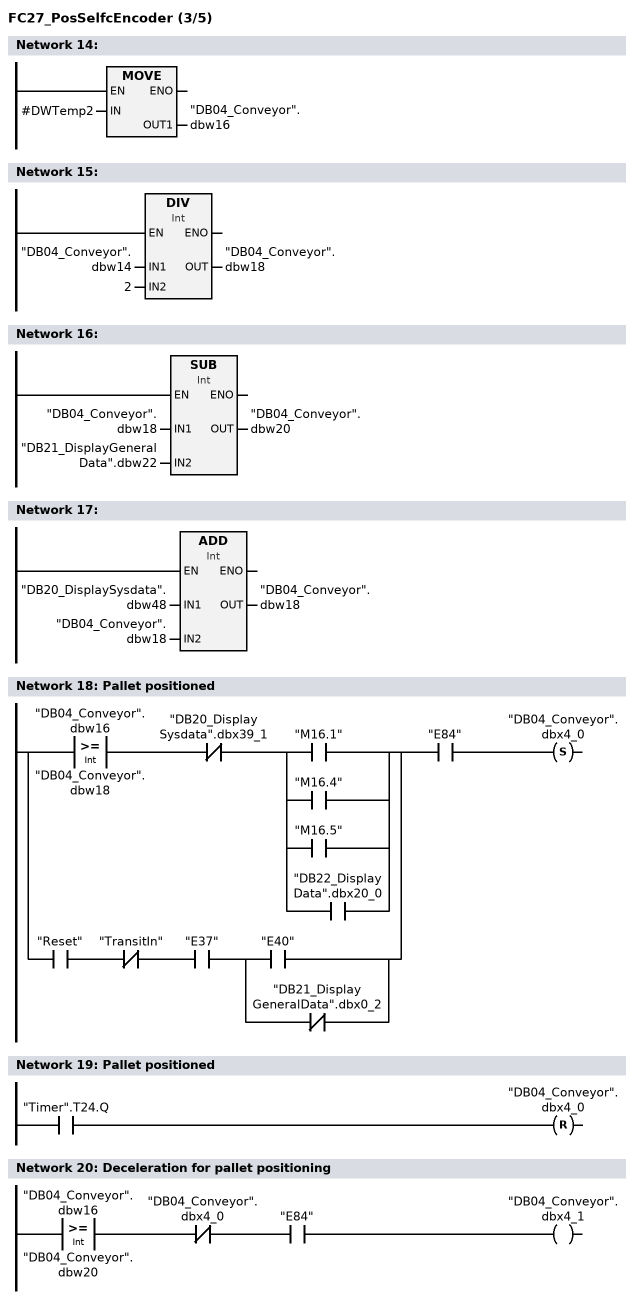
   RUNG wire#powerrail
      { S7_GenerateENO := "TRUE" } Move(in := #DWTemp2, out1 => "DB04_Conveyor".dbw16)
   END_RUNG
   // the same network as SCL:
   "DB04_Conveyor".dbw16 := #DWTemp2;
END_REGION

REGION Network 15
   RUNG wire#powerrail
      { S7_Templates := "SrcType := Int"; S7_GenerateENO := "TRUE" } Div(in1 := "DB04_Conveyor".dbw14, in2 := 2, out => "DB04_Conveyor".dbw18)
   END_RUNG
   // the same network as SCL:
   "DB04_Conveyor".dbw18 := "DB04_Conveyor".dbw14 / 2;
END_REGION

REGION Network 16
   RUNG wire#powerrail
      { S7_Templates := "SrcType := Int"; S7_GenerateENO := "TRUE" } Sub(in1 := "DB04_Conveyor".dbw18, in2 := "DB21_DisplayGeneralData".dbw22, out => "DB04_Conveyor".dbw20)
   END_RUNG
   // the same network as SCL:
   "DB04_Conveyor".dbw20 := "DB04_Conveyor".dbw18 - "DB21_DisplayGeneralData".dbw22;
END_REGION

REGION Network 17
   RUNG wire#powerrail
      { S7_Templates := "SrcType := Int"; S7_GenerateENO := "TRUE" } Add(in1 := "DB20_DisplaySysdata".dbw48, in2 := "DB04_Conveyor".dbw18, out => "DB04_Conveyor".dbw18)
   END_RUNG
   // the same network as SCL:
   "DB04_Conveyor".dbw18 := "DB20_DisplaySysdata".dbw48 + "DB04_Conveyor".dbw18;
END_REGION

REGION Network 18: Pallet positioned
   RUNG wire#powerrail
      { S7_Templates := "SrcType := Int" } GE_Contact(in1 := "DB04_Conveyor".dbw16, in2 := "DB04_Conveyor".dbw18)
      I_Contact( "DB20_DisplaySysdata".dbx39_1 )
      wire#w1
      Contact( "M16.1" )
      wire#w2
      Contact( "E84" )
      S_Coil( "DB04_Conveyor".dbx4_0 )
   END_RUNG
   RUNG wire#w1
      Contact( "M16.4" )
   END_RUNG wire#w2
   RUNG wire#w1
      Contact( "M16.5" )
   END_RUNG wire#w2
   RUNG wire#w1
      Contact( "DB22_DisplayData".dbx20_0 )
   END_RUNG wire#w2
   RUNG wire#powerrail
      Contact( "Reset" )
      I_Contact( "TransitIn" )
      Contact( "E37" )
      wire#w3
      Contact( "E40" )
   END_RUNG wire#w2
   RUNG wire#w3
      I_Contact( "DB21_DisplayGeneralData".dbx0_2 )
   END_RUNG wire#w2
   // the same network as SCL:
   IF ((("DB04_Conveyor".dbw16 >= "DB04_Conveyor".dbw18) AND NOT "DB20_DisplaySysdata".dbx39_1 AND ("M16.1" OR "M16.4" OR "M16.5" OR "DB22_DisplayData".dbx20_0)) OR ("Reset" AND NOT "TransitIn" AND "E37" AND ("E40" OR NOT "DB21_DisplayGeneralData".dbx0_2))) AND "E84" THEN
       "DB04_Conveyor".dbx4_0 := TRUE;
   END_IF;
END_REGION

REGION Network 19: Pallet positioned
   RUNG wire#powerrail
      Contact( "Timer".T24.Q )
      R_Coil( "DB04_Conveyor".dbx4_0 )
   END_RUNG
   // the same network as SCL:
   IF "Timer".T24.Q THEN "DB04_Conveyor".dbx4_0 := FALSE; END_IF;
END_REGION

REGION Network 20: Deceleration for pallet positioning
   RUNG wire#powerrail
      { S7_Templates := "SrcType := Int" } GE_Contact(in1 := "DB04_Conveyor".dbw16, in2 := "DB04_Conveyor".dbw20)
      I_Contact( "DB04_Conveyor".dbx4_0 )
      Contact( "E84" )
      Coil( "DB04_Conveyor".dbx4_1 )
   END_RUNG
   // the same network as SCL:
   "DB04_Conveyor".dbx4_1 := ("DB04_Conveyor".dbw16 >= "DB04_Conveyor".dbw20) AND NOT "DB04_Conveyor".dbx4_0 AND "E84";
END_REGION

REGION Network 21: Short pallet positioned
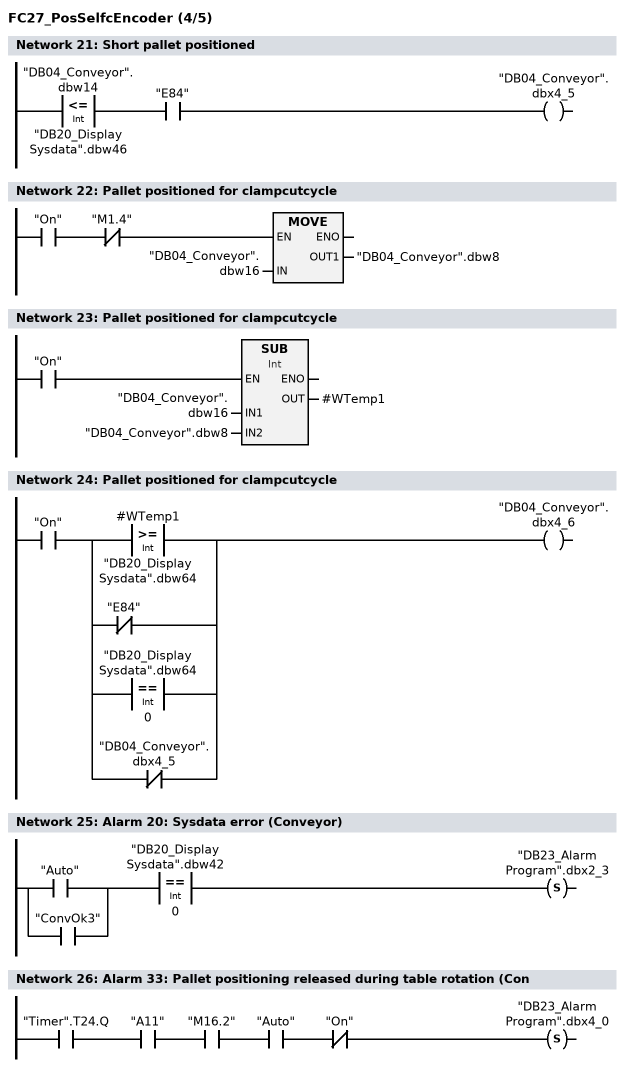
   RUNG wire#powerrail
      { S7_Templates := "SrcType := Int" } LE_Contact(in1 := "DB04_Conveyor".dbw14, in2 := "DB20_DisplaySysdata".dbw46)
      Contact( "E84" )
      Coil( "DB04_Conveyor".dbx4_5 )
   END_RUNG
   // the same network as SCL:
   "DB04_Conveyor".dbx4_5 := ("DB04_Conveyor".dbw14 <= "DB20_DisplaySysdata".dbw46) AND "E84";
END_REGION

REGION Network 22: Pallet positioned for clampcutcycle
   RUNG wire#powerrail
      Contact( "On" )
      I_Contact( "M1.4" )
      { S7_GenerateENO := "TRUE" } Move(in := "DB04_Conveyor".dbw16, out1 => "DB04_Conveyor".dbw8)
   END_RUNG
   // the same network as SCL:
   IF "On" AND NOT "M1.4" THEN "DB04_Conveyor".dbw8 := "DB04_Conveyor".dbw16; END_IF;
END_REGION

REGION Network 23: Pallet positioned for clampcutcycle
   RUNG wire#powerrail
      Contact( "On" )
      { S7_Templates := "SrcType := Int"; S7_GenerateENO := "TRUE" } Sub(in1 := "DB04_Conveyor".dbw16, in2 := "DB04_Conveyor".dbw8, out => #WTemp1)
   END_RUNG
   // the same network as SCL:
   IF "On" THEN #WTemp1 := "DB04_Conveyor".dbw16 - "DB04_Conveyor".dbw8; END_IF;
END_REGION

REGION Network 24: Pallet positioned for clampcutcycle
   RUNG wire#powerrail
      Contact( "On" )
      wire#w1
      { S7_Templates := "SrcType := Int" } GE_Contact(in1 := #WTemp1, in2 := "DB20_DisplaySysdata".dbw64)
      wire#w2
      Coil( "DB04_Conveyor".dbx4_6 )
   END_RUNG
   RUNG wire#w1
      I_Contact( "E84" )
   END_RUNG wire#w2
   RUNG wire#w1
      { S7_Templates := "SrcType := Int" } EQ_Contact(in1 := "DB20_DisplaySysdata".dbw64, in2 := 0)
   END_RUNG wire#w2
   RUNG wire#w1
      I_Contact( "DB04_Conveyor".dbx4_5 )
   END_RUNG wire#w2
   // the same network as SCL:
   "DB04_Conveyor".dbx4_6 := "On" AND ((#WTemp1 >= "DB20_DisplaySysdata".dbw64) OR NOT "E84" OR ("DB20_DisplaySysdata".dbw64 = 0) OR NOT "DB04_Conveyor".dbx4_5);
END_REGION

REGION Network 25: Alarm 20: Sysdata error (Conveyor)
   RUNG wire#powerrail
      Contact( "Auto" )
      wire#w1
      { S7_Templates := "SrcType := Int" } EQ_Contact(in1 := "DB20_DisplaySysdata".dbw42, in2 := 0)
      S_Coil( "DB23_AlarmProgram".dbx2_3 )
   END_RUNG
   RUNG wire#powerrail
      Contact( "ConvOk3" )
   END_RUNG wire#w1
   // the same network as SCL:
   IF ("Auto" OR "ConvOk3") AND ("DB20_DisplaySysdata".dbw42 = 0) THEN
       "DB23_AlarmProgram".dbx2_3 := TRUE;
   END_IF;
END_REGION

REGION Network 26: Alarm 33: Pallet positioning released during table rotation (Con
   RUNG wire#powerrail
      Contact( "Timer".T24.Q )
      Contact( "A11" )
      Contact( "M16.2" )
      Contact( "Auto" )
      I_Contact( "On" )
      S_Coil( "DB23_AlarmProgram".dbx4_0 )
   END_RUNG
   // the same network as SCL:
   IF "Timer".T24.Q AND "A11" AND "M16.2" AND "Auto" AND NOT "On" THEN
       "DB23_AlarmProgram".dbx4_0 := TRUE;
   END_IF;
END_REGION

REGION Network 27: Alarm 36: Wrong pallet positioning (Conveyor)
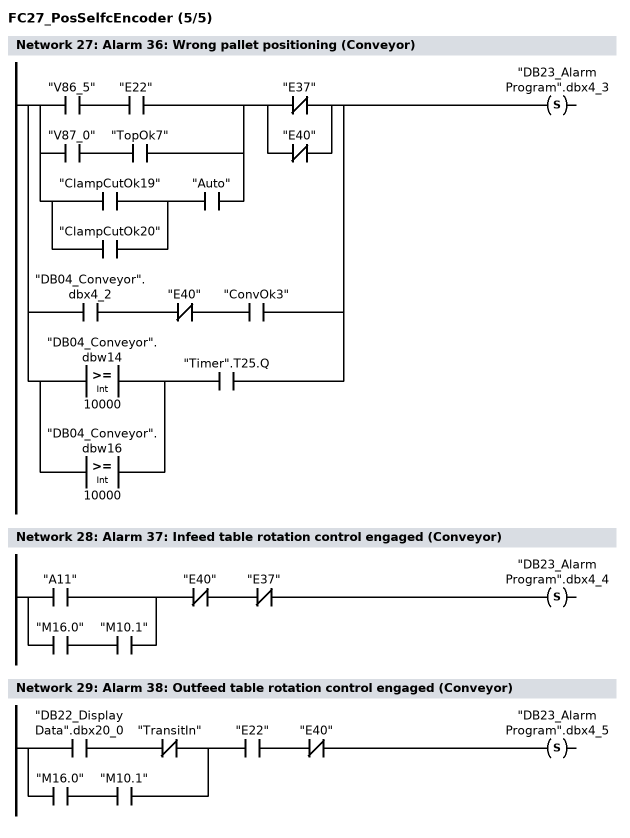
   RUNG wire#powerrail
      Contact( "V86_5" )
      Contact( "E22" )
      wire#w1
      I_Contact( "E37" )
      wire#w3
      S_Coil( "DB23_AlarmProgram".dbx4_3 )
   END_RUNG
   RUNG wire#powerrail
      Contact( "V87_0" )
      Contact( "TopOk7" )
   END_RUNG wire#w1
   RUNG wire#powerrail
      Contact( "ClampCutOk19" )
      wire#w2
      Contact( "Auto" )
   END_RUNG wire#w1
   RUNG wire#powerrail
      Contact( "ClampCutOk20" )
   END_RUNG wire#w2
   RUNG wire#w1
      I_Contact( "E40" )
   END_RUNG wire#w3
   RUNG wire#powerrail
      Contact( "DB04_Conveyor".dbx4_2 )
      I_Contact( "E40" )
      Contact( "ConvOk3" )
   END_RUNG wire#w3
   RUNG wire#powerrail
      { S7_Templates := "SrcType := Int" } GE_Contact(in1 := "DB04_Conveyor".dbw14, in2 := 10000)
      wire#w4
      Contact( "Timer".T25.Q )
   END_RUNG wire#w3
   RUNG wire#powerrail
      { S7_Templates := "SrcType := Int" } GE_Contact(in1 := "DB04_Conveyor".dbw16, in2 := 10000)
   END_RUNG wire#w4
   // the same network as SCL:
   IF ((("V86_5" AND "E22") OR ("V87_0" AND "TopOk7") OR (("ClampCutOk19" OR "ClampCutOk20") AND "Auto")) AND (NOT "E37" OR NOT "E40")) OR ("DB04_Conveyor".dbx4_2 AND NOT "E40" AND "ConvOk3") OR ((("DB04_Conveyor".dbw14 >= 10000) OR ("DB04_Conveyor".dbw16 >= 10000)) AND "Timer".T25.Q) THEN
       "DB23_AlarmProgram".dbx4_3 := TRUE;
   END_IF;
END_REGION

REGION Network 28: Alarm 37: Infeed table rotation control engaged (Conveyor)
   RUNG wire#powerrail
      Contact( "A11" )
      wire#w1
      I_Contact( "E40" )
      I_Contact( "E37" )
      S_Coil( "DB23_AlarmProgram".dbx4_4 )
   END_RUNG
   RUNG wire#powerrail
      Contact( "M16.0" )
      Contact( "M10.1" )
   END_RUNG wire#w1
   // the same network as SCL:
   IF ("A11" OR ("M16.0" AND "M10.1")) AND NOT "E40" AND NOT "E37" THEN
       "DB23_AlarmProgram".dbx4_4 := TRUE;
   END_IF;
END_REGION

REGION Network 29: Alarm 38: Outfeed table rotation control engaged (Conveyor)
   RUNG wire#powerrail
      Contact( "DB22_DisplayData".dbx20_0 )
      I_Contact( "TransitIn" )
      wire#w1
      Contact( "E22" )
      I_Contact( "E40" )
      S_Coil( "DB23_AlarmProgram".dbx4_5 )
   END_RUNG
   RUNG wire#powerrail
      Contact( "M16.0" )
      Contact( "M10.1" )
   END_RUNG wire#w1
   // the same network as SCL:
   IF (("DB22_DisplayData".dbx20_0 AND NOT "TransitIn") OR ("M16.0" AND "M10.1")) AND "E22" AND NOT "E40" THEN
       "DB23_AlarmProgram".dbx4_5 := TRUE;
   END_IF;
END_REGION
END_FUNCTION

FUNCTION "FC31_ConveyorInverter" : Void   // FC31, LAD
TITLE = Conveyor management with inverter
{ S7_Optimized_Access := 'FALSE' }
AUTHOR : Robopac
VERSION : 0.0
// stored: AutoNumber false, IsIECCheckEnabled false, SetENOAutomatically false, UDAEnableTagReadback false
   VAR_TEMP
      TimeUpwardTableCycle : Word;
      TimeUpwardTableCycleInt : Int;
      TempWord : Word;
   END_VAR
   VAR_TEMP   // added for the SCL form of the ladder/FBD networks
      _w1 : Bool;
   END_VAR
BEGIN

REGION Network 1: Timer SA type for conveyor motor
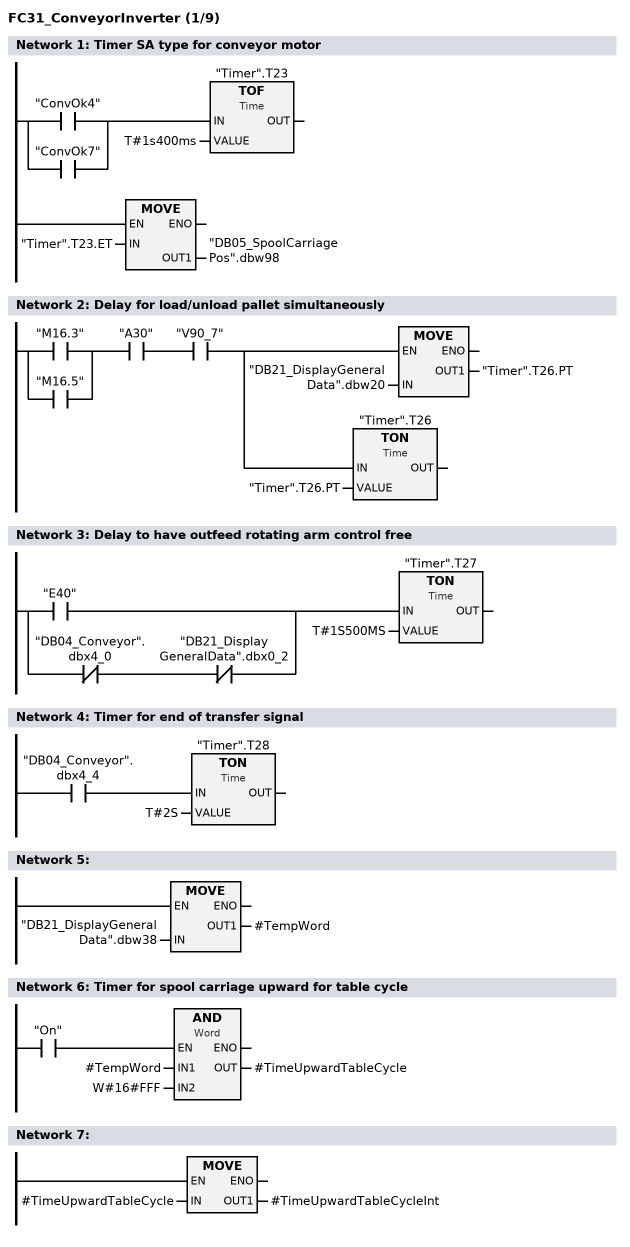
   "Timer".T23.TOF(IN := "ConvOk4" OR "ConvOk7", PT := T#1s400ms);   // TOF coil
   "DB05_SpoolCarriagePos".dbw98 := "Timer".T23.ET;
END_REGION

REGION Network 2: Delay for load/unload pallet simultaneously
   #_w1 := ("M16.3" OR "M16.5") AND "A30" AND "V90_7";
   IF #_w1 THEN "Timer".T26.PT := "DB21_DisplayGeneralData".dbw20; END_IF;
   "Timer".T26.TON(IN := #_w1, PT := "Timer".T26.PT);   // TON coil
END_REGION

REGION Network 3: Delay to have outfeed rotating arm control free
   "Timer".T27.TON(IN := "E40" OR (NOT "DB04_Conveyor".dbx4_0 AND NOT "DB21_DisplayGeneralData".dbx0_2), PT := T#1S500MS);   // TON coil
END_REGION

REGION Network 4: Timer for end of transfer signal
   "Timer".T28.TON(IN := "DB04_Conveyor".dbx4_4, PT := T#2S);   // TON coil
END_REGION

REGION Network 5
   RUNG wire#powerrail
      { S7_GenerateENO := "TRUE" } Move(in := "DB21_DisplayGeneralData".dbw38, out1 => #TempWord)
   END_RUNG
   // the same network as SCL:
   #TempWord := "DB21_DisplayGeneralData".dbw38;
END_REGION

REGION Network 6: Timer for spool carriage upward for table cycle
   RUNG wire#powerrail
      Contact( "On" )
      { S7_Templates := "SrcType := Word"; S7_GenerateENO := "TRUE" } And(in1 := #TempWord, in2 := W#16#FFF, out => #TimeUpwardTableCycle)
   END_RUNG
   // the same network as SCL:
   IF "On" THEN #TimeUpwardTableCycle := #TempWord AND W#16#FFF; END_IF;
END_REGION

REGION Network 7
   RUNG wire#powerrail
      { S7_GenerateENO := "TRUE" } Move(in := #TimeUpwardTableCycle, out1 => #TimeUpwardTableCycleInt)
   END_RUNG
   // the same network as SCL:
   #TimeUpwardTableCycleInt := #TimeUpwardTableCycle;
END_REGION

REGION Network 8: Timer for spool carriage upward for table cycle
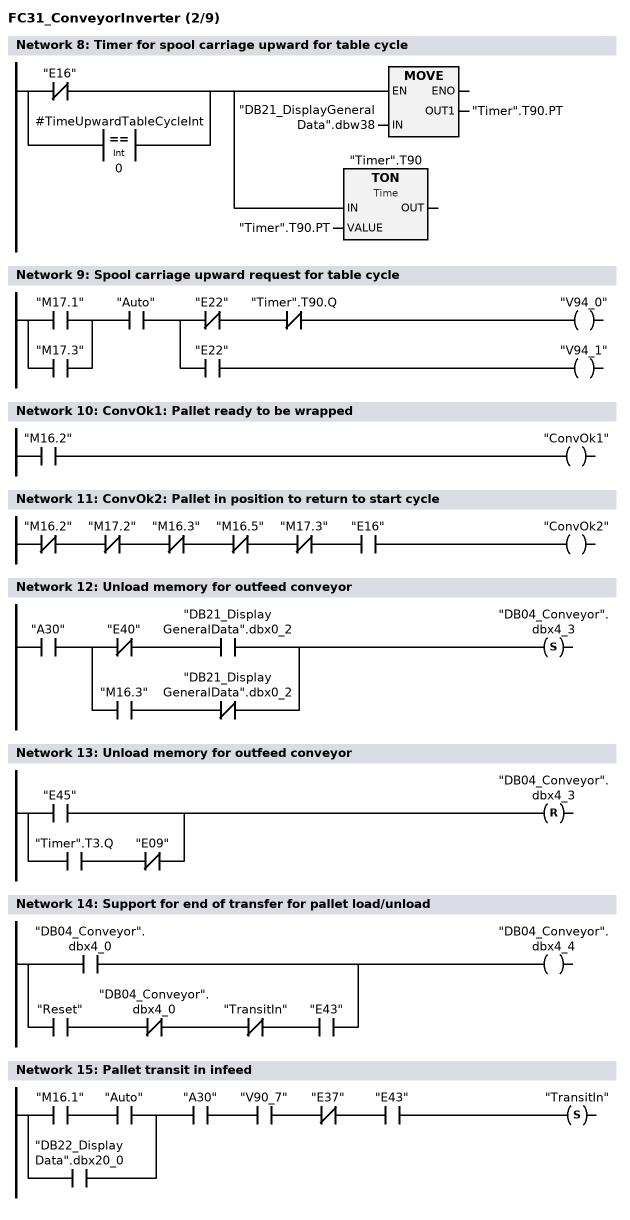
   #_w1 := NOT "E16" OR (#TimeUpwardTableCycleInt = 0);
   IF #_w1 THEN "Timer".T90.PT := "DB21_DisplayGeneralData".dbw38; END_IF;
   "Timer".T90.TON(IN := #_w1, PT := "Timer".T90.PT);   // TON coil
END_REGION

REGION Network 9: Spool carriage upward request for table cycle
   RUNG wire#powerrail
      Contact( "M17.1" )
      wire#w1
      Contact( "Auto" )
      wire#w2
      I_Contact( "E22" )
      I_Contact( "Timer".T90.Q )
      Coil( "V94_0" )
   END_RUNG
   RUNG wire#powerrail
      Contact( "M17.3" )
   END_RUNG wire#w1
   RUNG wire#w2
      Contact( "E22" )
      Coil( "V94_1" )
   END_RUNG
   // the same network as SCL:
   #_w1 := ("M17.1" OR "M17.3") AND "Auto";
   "V94_0" := #_w1 AND NOT "E22" AND NOT "Timer".T90.Q;
   "V94_1" := #_w1 AND "E22";
END_REGION

REGION Network 10: ConvOk1: Pallet ready to be wrapped
   RUNG wire#powerrail
      Contact( "M16.2" )
      Coil( "ConvOk1" )
   END_RUNG
   // the same network as SCL:
   "ConvOk1" := "M16.2";
END_REGION

REGION Network 11: ConvOk2: Pallet in position to return to start cycle
   RUNG wire#powerrail
      I_Contact( "M16.2" )
      I_Contact( "M17.2" )
      I_Contact( "M16.3" )
      I_Contact( "M16.5" )
      I_Contact( "M17.3" )
      Contact( "E16" )
      Coil( "ConvOk2" )
   END_RUNG
   // the same network as SCL:
   "ConvOk2" := NOT "M16.2" AND NOT "M17.2" AND NOT "M16.3" AND NOT "M16.5" AND NOT "M17.3" AND "E16";
END_REGION

REGION Network 12: Unload memory for outfeed conveyor
   RUNG wire#powerrail
      Contact( "A30" )
      wire#w1
      I_Contact( "E40" )
      Contact( "DB21_DisplayGeneralData".dbx0_2 )
      wire#w2
      S_Coil( "DB04_Conveyor".dbx4_3 )
   END_RUNG
   RUNG wire#w1
      Contact( "M16.3" )
      I_Contact( "DB21_DisplayGeneralData".dbx0_2 )
   END_RUNG wire#w2
   // the same network as SCL:
   IF "A30" AND ((NOT "E40" AND "DB21_DisplayGeneralData".dbx0_2) OR ("M16.3" AND NOT "DB21_DisplayGeneralData".dbx0_2)) THEN
       "DB04_Conveyor".dbx4_3 := TRUE;
   END_IF;
END_REGION

REGION Network 13: Unload memory for outfeed conveyor
   RUNG wire#powerrail
      Contact( "E45" )
      wire#w1
      R_Coil( "DB04_Conveyor".dbx4_3 )
   END_RUNG
   RUNG wire#powerrail
      Contact( "Timer".T3.Q )
      I_Contact( "E09" )
   END_RUNG wire#w1
   // the same network as SCL:
   IF "E45" OR ("Timer".T3.Q AND NOT "E09") THEN "DB04_Conveyor".dbx4_3 := FALSE; END_IF;
END_REGION

REGION Network 14: Support for end of transfer for pallet load/unload
   RUNG wire#powerrail
      Contact( "DB04_Conveyor".dbx4_0 )
      wire#w1
      Coil( "DB04_Conveyor".dbx4_4 )
   END_RUNG
   RUNG wire#powerrail
      Contact( "Reset" )
      I_Contact( "DB04_Conveyor".dbx4_0 )
      I_Contact( "TransitIn" )
      Contact( "E43" )
   END_RUNG wire#w1
   // the same network as SCL:
   "DB04_Conveyor".dbx4_4 := "DB04_Conveyor".dbx4_0 OR ("Reset" AND NOT "DB04_Conveyor".dbx4_0 AND NOT "TransitIn" AND "E43");
END_REGION

REGION Network 15: Pallet transit in infeed
   RUNG wire#powerrail
      Contact( "M16.1" )
      Contact( "Auto" )
      wire#w1
      Contact( "A30" )
      Contact( "V90_7" )
      I_Contact( "E37" )
      Contact( "E43" )
      S_Coil( "TransitIn" )
   END_RUNG
   RUNG wire#powerrail
      Contact( "DB22_DisplayData".dbx20_0 )
   END_RUNG wire#w1
   // the same network as SCL:
   IF (("M16.1" AND "Auto") OR "DB22_DisplayData".dbx20_0) AND "A30" AND "V90_7" AND NOT "E37" AND "E43" THEN
       "TransitIn" := TRUE;
   END_IF;
END_REGION

REGION Network 16: Pallet transit in infeed
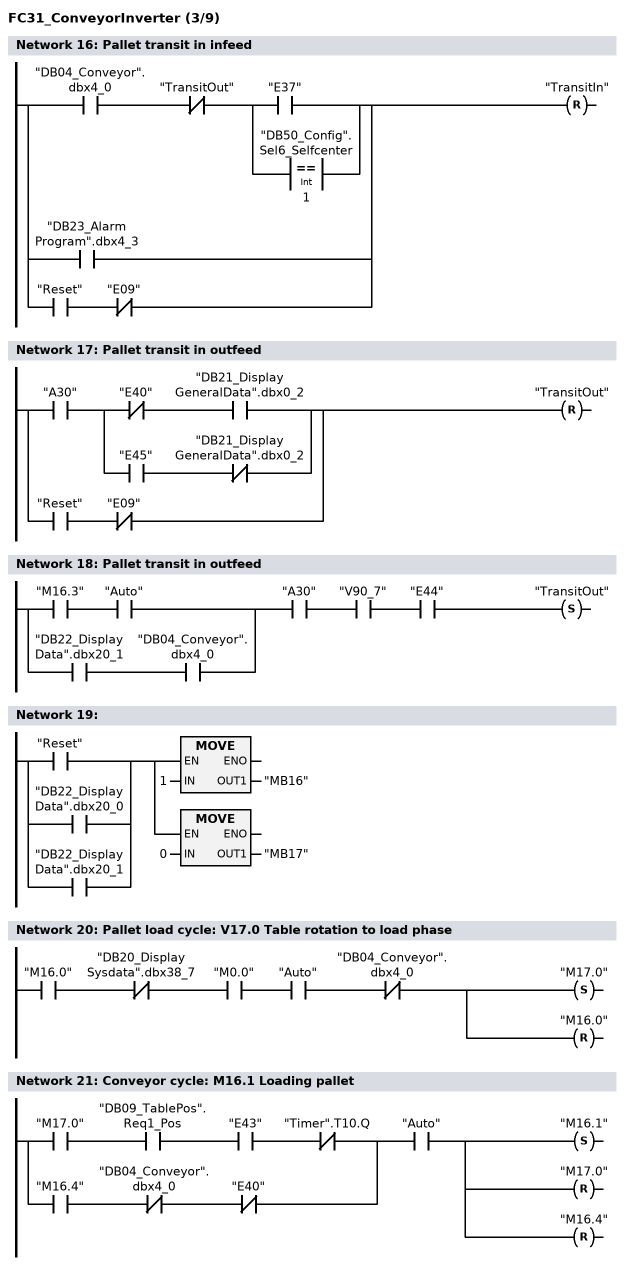
   IF ("DB04_Conveyor".dbx4_0 AND NOT "TransitOut" AND (("DB50_Config".Sel6_Selfcenter = 1) OR "E37")) OR "DB23_AlarmProgram".dbx4_3 OR ("Reset" AND NOT "E09") THEN
       "TransitIn" := FALSE;
   END_IF;
END_REGION

REGION Network 17: Pallet transit in outfeed
   RUNG wire#powerrail
      Contact( "A30" )
      wire#w1
      I_Contact( "E40" )
      Contact( "DB21_DisplayGeneralData".dbx0_2 )
      wire#w2
      R_Coil( "TransitOut" )
   END_RUNG
   RUNG wire#w1
      Contact( "E45" )
      I_Contact( "DB21_DisplayGeneralData".dbx0_2 )
   END_RUNG wire#w2
   RUNG wire#powerrail
      Contact( "Reset" )
      I_Contact( "E09" )
   END_RUNG wire#w2
   // the same network as SCL:
   IF ("A30" AND ((NOT "E40" AND "DB21_DisplayGeneralData".dbx0_2) OR ("E45" AND NOT "DB21_DisplayGeneralData".dbx0_2))) OR ("Reset" AND NOT "E09") THEN
       "TransitOut" := FALSE;
   END_IF;
END_REGION

REGION Network 18: Pallet transit in outfeed
   RUNG wire#powerrail
      Contact( "M16.3" )
      Contact( "Auto" )
      wire#w1
      Contact( "A30" )
      Contact( "V90_7" )
      Contact( "E44" )
      S_Coil( "TransitOut" )
   END_RUNG
   RUNG wire#powerrail
      Contact( "DB22_DisplayData".dbx20_1 )
      Contact( "DB04_Conveyor".dbx4_0 )
   END_RUNG wire#w1
   // the same network as SCL:
   IF (("M16.3" AND "Auto") OR ("DB22_DisplayData".dbx20_1 AND "DB04_Conveyor".dbx4_0)) AND "A30" AND "V90_7" AND "E44" THEN
       "TransitOut" := TRUE;
   END_IF;
END_REGION

REGION Network 19
   RUNG wire#powerrail
      Contact( "Reset" )
      wire#w1
      { S7_GenerateENO := "TRUE" } Move(in := 1, out1 => "MB16")
   END_RUNG
   RUNG wire#powerrail
      Contact( "DB22_DisplayData".dbx20_0 )
   END_RUNG wire#w1
   RUNG wire#powerrail
      Contact( "DB22_DisplayData".dbx20_1 )
   END_RUNG wire#w1
   RUNG wire#w1
      { S7_GenerateENO := "TRUE" } Move(in := 0, out1 => "MB17")
   END_RUNG
   // the same network as SCL:
   IF "Reset" OR "DB22_DisplayData".dbx20_0 OR "DB22_DisplayData".dbx20_1 THEN
       "MB16" := 1;
       "MB17" := 0;
   END_IF;
END_REGION

REGION Network 20: Pallet load cycle: V17.0 Table rotation to load phase
   RUNG wire#powerrail
      Contact( "M16.0" )
      I_Contact( "DB20_DisplaySysdata".dbx38_7 )
      Contact( "M0.0" )
      Contact( "Auto" )
      I_Contact( "DB04_Conveyor".dbx4_0 )
      wire#w1
      S_Coil( "M17.0" )
   END_RUNG
   RUNG wire#w1
      R_Coil( "M16.0" )
   END_RUNG
   // the same network as SCL:
   IF "M16.0" AND NOT "DB20_DisplaySysdata".dbx38_7 AND "M0.0" AND "Auto" AND NOT "DB04_Conveyor".dbx4_0 THEN
       "M17.0" := TRUE;
       "M16.0" := FALSE;
   END_IF;
END_REGION

REGION Network 21: Conveyor cycle: M16.1 Loading pallet
   RUNG wire#powerrail
      Contact( "M17.0" )
      Contact( "DB09_TablePos".Req1_Pos )
      Contact( "E43" )
      I_Contact( "Timer".T10.Q )
      wire#w1
      Contact( "Auto" )
      wire#w2
      S_Coil( "M16.1" )
   END_RUNG
   RUNG wire#powerrail
      Contact( "M16.4" )
      I_Contact( "DB04_Conveyor".dbx4_0 )
      I_Contact( "E40" )
   END_RUNG wire#w1
   RUNG wire#w2
      R_Coil( "M17.0" )
   END_RUNG
   RUNG wire#w2
      R_Coil( "M16.4" )
   END_RUNG
   // the same network as SCL:
   IF (("M17.0" AND "DB09_TablePos".Req1_Pos AND "E43" AND NOT "Timer".T10.Q) OR ("M16.4" AND NOT "DB04_Conveyor".dbx4_0 AND NOT "E40")) AND "Auto" THEN
       "M16.1" := TRUE;
   END_IF;
   #_w1 := (("M17.0" AND "DB09_TablePos".Req1_Pos AND "E43" AND NOT "Timer".T10.Q) OR ("M16.4" AND NOT "DB04_Conveyor".dbx4_0 AND NOT "E40")) AND "Auto";
   IF #_w1 THEN
       "M17.0" := FALSE;
       "M16.4" := FALSE;
   END_IF;
END_REGION

REGION Network 22: Pallet load cycle: V17.1 Table rotation to machine phase from lo
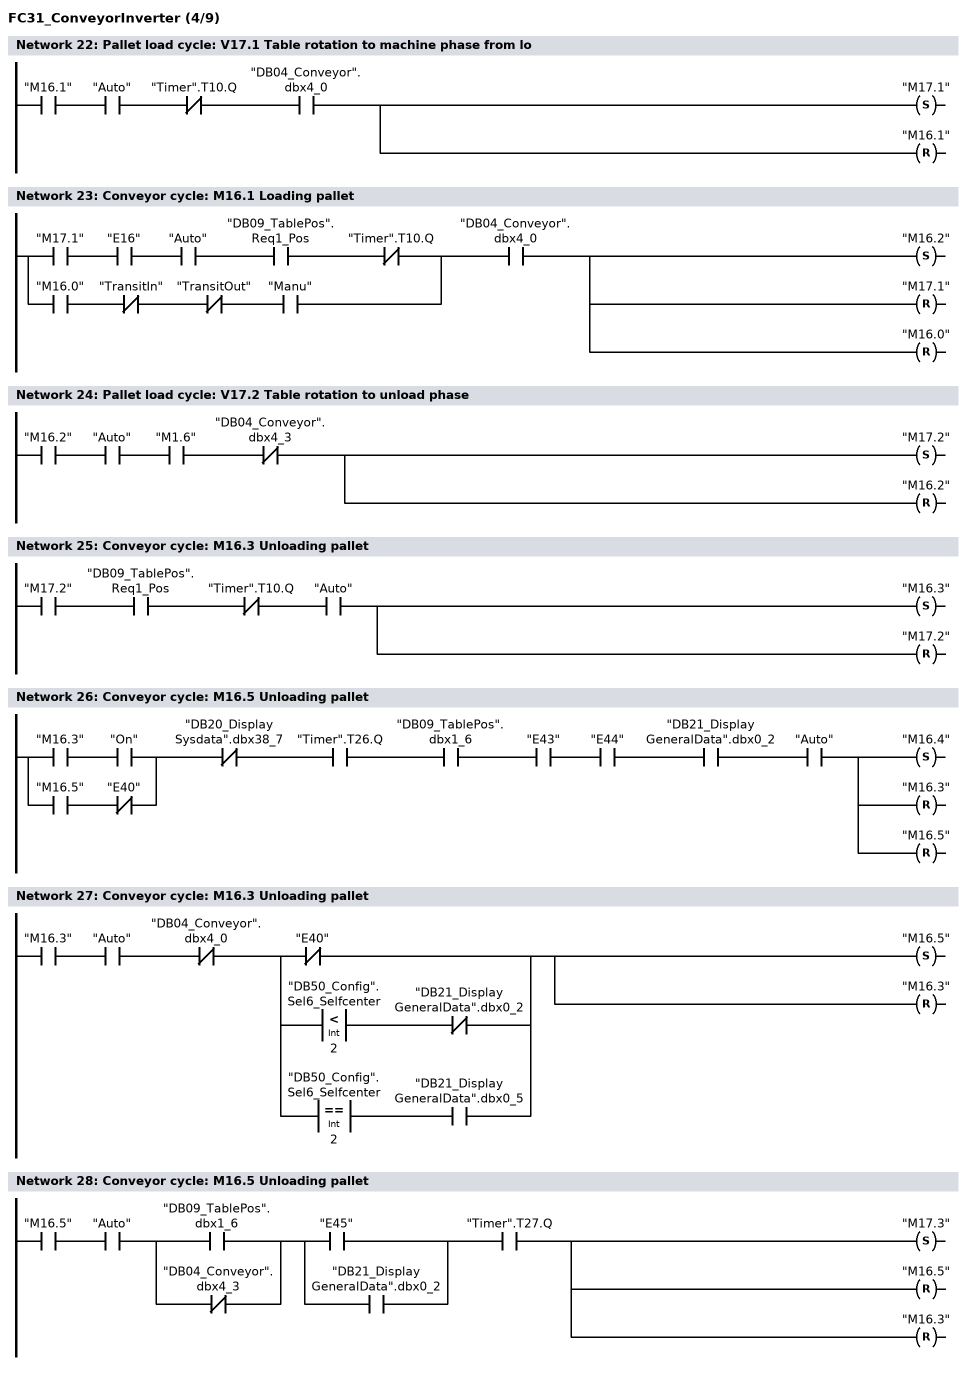
   RUNG wire#powerrail
      Contact( "M16.1" )
      Contact( "Auto" )
      I_Contact( "Timer".T10.Q )
      Contact( "DB04_Conveyor".dbx4_0 )
      wire#w1
      S_Coil( "M17.1" )
   END_RUNG
   RUNG wire#w1
      R_Coil( "M16.1" )
   END_RUNG
   // the same network as SCL:
   IF "M16.1" AND "Auto" AND NOT "Timer".T10.Q AND "DB04_Conveyor".dbx4_0 THEN
       "M17.1" := TRUE;
       "M16.1" := FALSE;
   END_IF;
END_REGION

REGION Network 23: Conveyor cycle: M16.1 Loading pallet
   RUNG wire#powerrail
      Contact( "M17.1" )
      Contact( "E16" )
      Contact( "Auto" )
      Contact( "DB09_TablePos".Req1_Pos )
      I_Contact( "Timer".T10.Q )
      wire#w1
      Contact( "DB04_Conveyor".dbx4_0 )
      wire#w2
      S_Coil( "M16.2" )
   END_RUNG
   RUNG wire#powerrail
      Contact( "M16.0" )
      I_Contact( "TransitIn" )
      I_Contact( "TransitOut" )
      Contact( "Manu" )
   END_RUNG wire#w1
   RUNG wire#w2
      R_Coil( "M17.1" )
   END_RUNG
   RUNG wire#w2
      R_Coil( "M16.0" )
   END_RUNG
   // the same network as SCL:
   IF (("M17.1" AND "E16" AND "Auto" AND "DB09_TablePos".Req1_Pos AND NOT "Timer".T10.Q) OR ("M16.0" AND NOT "TransitIn" AND NOT "TransitOut" AND "Manu")) AND "DB04_Conveyor".dbx4_0 THEN
       "M16.2" := TRUE;
   END_IF;
   #_w1 := (("M17.1" AND "E16" AND "Auto" AND "DB09_TablePos".Req1_Pos AND NOT "Timer".T10.Q) OR ("M16.0" AND NOT "TransitIn" AND NOT "TransitOut" AND "Manu")) AND "DB04_Conveyor".dbx4_0;
   IF #_w1 THEN
       "M17.1" := FALSE;
       "M16.0" := FALSE;
   END_IF;
END_REGION

REGION Network 24: Pallet load cycle: V17.2 Table rotation to unload phase
   RUNG wire#powerrail
      Contact( "M16.2" )
      Contact( "Auto" )
      Contact( "M1.6" )
      I_Contact( "DB04_Conveyor".dbx4_3 )
      wire#w1
      S_Coil( "M17.2" )
   END_RUNG
   RUNG wire#w1
      R_Coil( "M16.2" )
   END_RUNG
   // the same network as SCL:
   IF "M16.2" AND "Auto" AND "M1.6" AND NOT "DB04_Conveyor".dbx4_3 THEN
       "M17.2" := TRUE;
       "M16.2" := FALSE;
   END_IF;
END_REGION

REGION Network 25: Conveyor cycle: M16.3 Unloading pallet
   RUNG wire#powerrail
      Contact( "M17.2" )
      Contact( "DB09_TablePos".Req1_Pos )
      I_Contact( "Timer".T10.Q )
      Contact( "Auto" )
      wire#w1
      S_Coil( "M16.3" )
   END_RUNG
   RUNG wire#w1
      R_Coil( "M17.2" )
   END_RUNG
   // the same network as SCL:
   IF "M17.2" AND "DB09_TablePos".Req1_Pos AND NOT "Timer".T10.Q AND "Auto" THEN
       "M16.3" := TRUE;
       "M17.2" := FALSE;
   END_IF;
END_REGION

REGION Network 26: Conveyor cycle: M16.5 Unloading pallet
   RUNG wire#powerrail
      Contact( "M16.3" )
      Contact( "On" )
      wire#w1
      I_Contact( "DB20_DisplaySysdata".dbx38_7 )
      Contact( "Timer".T26.Q )
      Contact( "DB09_TablePos".dbx1_6 )
      Contact( "E43" )
      Contact( "E44" )
      Contact( "DB21_DisplayGeneralData".dbx0_2 )
      Contact( "Auto" )
      wire#w2
      S_Coil( "M16.4" )
   END_RUNG
   RUNG wire#powerrail
      Contact( "M16.5" )
      I_Contact( "E40" )
   END_RUNG wire#w1
   RUNG wire#w2
      R_Coil( "M16.3" )
   END_RUNG
   RUNG wire#w2
      R_Coil( "M16.5" )
   END_RUNG
   // the same network as SCL:
   IF (("M16.3" AND "On") OR ("M16.5" AND NOT "E40")) AND NOT "DB20_DisplaySysdata".dbx38_7 AND "Timer".T26.Q AND "DB09_TablePos".dbx1_6 AND "E43" AND "E44" AND "DB21_DisplayGeneralData".dbx0_2 AND "Auto" THEN
       "M16.4" := TRUE;
   END_IF;
   #_w1 := (("M16.3" AND "On") OR ("M16.5" AND NOT "E40")) AND NOT "DB20_DisplaySysdata".dbx38_7 AND "Timer".T26.Q AND "DB09_TablePos".dbx1_6 AND "E43" AND "E44" AND "DB21_DisplayGeneralData".dbx0_2 AND "Auto";
   IF #_w1 THEN
       "M16.3" := FALSE;
       "M16.5" := FALSE;
   END_IF;
END_REGION

REGION Network 27: Conveyor cycle: M16.3 Unloading pallet
   RUNG wire#powerrail
      Contact( "M16.3" )
      Contact( "Auto" )
      I_Contact( "DB04_Conveyor".dbx4_0 )
      wire#w1
      I_Contact( "E40" )
      wire#w2
      S_Coil( "M16.5" )
   END_RUNG
   RUNG wire#w1
      { S7_Templates := "SrcType := Int" } LT_Contact(in1 := "DB50_Config".Sel6_Selfcenter, in2 := 2)
      I_Contact( "DB21_DisplayGeneralData".dbx0_2 )
   END_RUNG wire#w2
   RUNG wire#w1
      { S7_Templates := "SrcType := Int" } EQ_Contact(in1 := "DB50_Config".Sel6_Selfcenter, in2 := 2)
      Contact( "DB21_DisplayGeneralData".dbx0_5 )
   END_RUNG wire#w2
   RUNG wire#w2
      R_Coil( "M16.3" )
   END_RUNG
   // the same network as SCL:
   IF "M16.3" AND "Auto" AND NOT "DB04_Conveyor".dbx4_0 AND (NOT "E40" OR (("DB50_Config".Sel6_Selfcenter < 2) AND NOT "DB21_DisplayGeneralData".dbx0_2) OR (("DB50_Config".Sel6_Selfcenter = 2) AND "DB21_DisplayGeneralData".dbx0_5)) THEN
       "M16.5" := TRUE;
       "M16.3" := FALSE;
   END_IF;
END_REGION

REGION Network 28: Conveyor cycle: M16.5 Unloading pallet
   RUNG wire#powerrail
      Contact( "M16.5" )
      Contact( "Auto" )
      wire#w1
      Contact( "DB09_TablePos".dbx1_6 )
      wire#w2
      Contact( "E45" )
      wire#w3
      Contact( "Timer".T27.Q )
      wire#w4
      S_Coil( "M17.3" )
   END_RUNG
   RUNG wire#w1
      I_Contact( "DB04_Conveyor".dbx4_3 )
   END_RUNG wire#w2
   RUNG wire#w2
      Contact( "DB21_DisplayGeneralData".dbx0_2 )
   END_RUNG wire#w3
   RUNG wire#w4
      R_Coil( "M16.5" )
   END_RUNG
   RUNG wire#w4
      R_Coil( "M16.3" )
   END_RUNG
   // the same network as SCL:
   IF "M16.5" AND "Auto" AND ("DB09_TablePos".dbx1_6 OR NOT "DB04_Conveyor".dbx4_3) AND ("E45" OR "DB21_DisplayGeneralData".dbx0_2) AND "Timer".T27.Q THEN
       "M17.3" := TRUE;
   END_IF;
   #_w1 := "M16.5" AND "Auto" AND ("DB09_TablePos".dbx1_6 OR NOT "DB04_Conveyor".dbx4_3) AND ("E45" OR "DB21_DisplayGeneralData".dbx0_2) AND "Timer".T27.Q;
   IF #_w1 THEN
       "M16.5" := FALSE;
       "M16.3" := FALSE;
   END_IF;
END_REGION

REGION Network 29: Conveyor cycle: M16.0 Start cycle
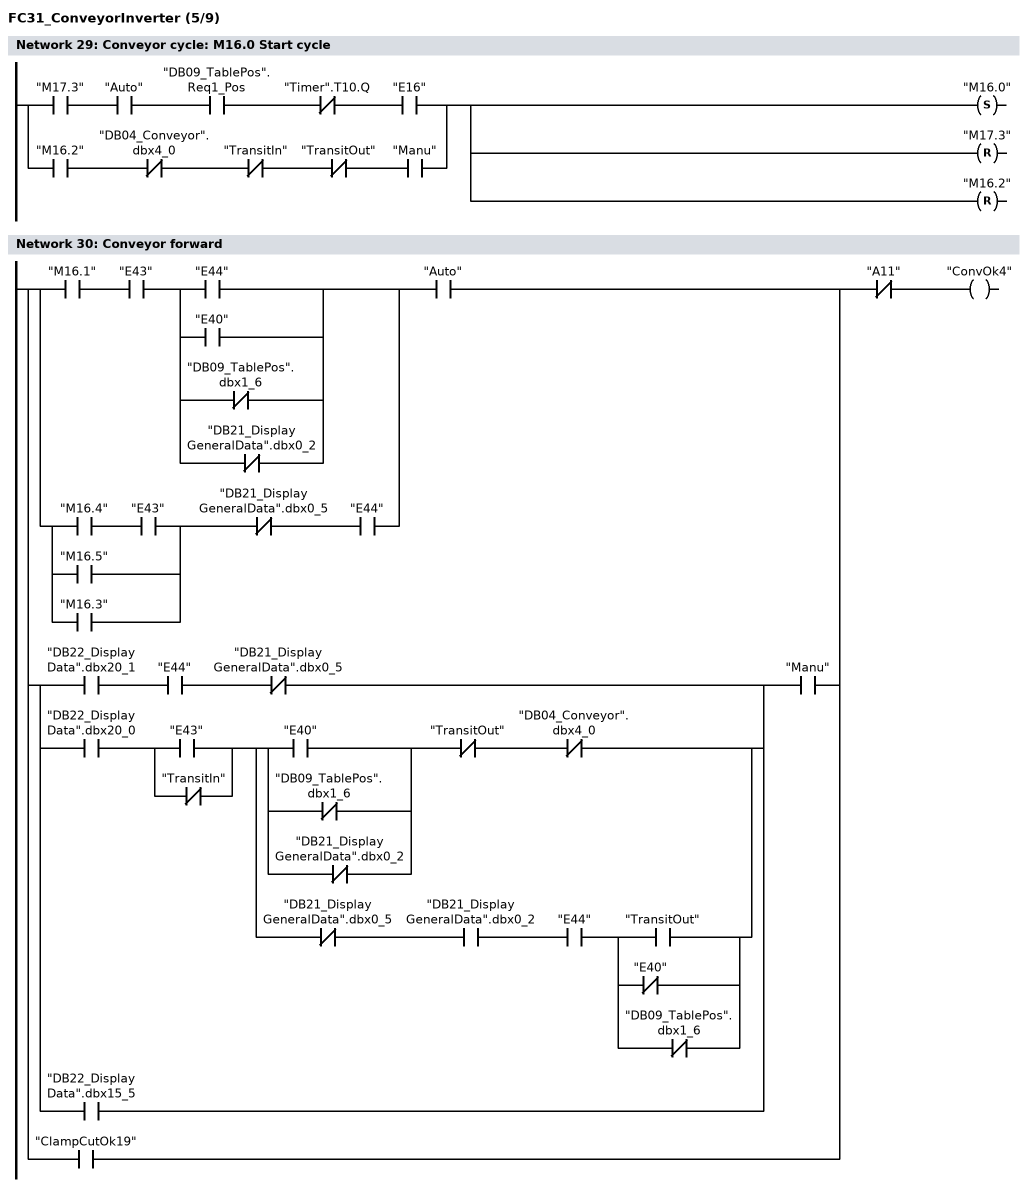
   RUNG wire#powerrail
      Contact( "M17.3" )
      Contact( "Auto" )
      Contact( "DB09_TablePos".Req1_Pos )
      I_Contact( "Timer".T10.Q )
      Contact( "E16" )
      wire#w1
      S_Coil( "M16.0" )
   END_RUNG
   RUNG wire#powerrail
      Contact( "M16.2" )
      I_Contact( "DB04_Conveyor".dbx4_0 )
      I_Contact( "TransitIn" )
      I_Contact( "TransitOut" )
      Contact( "Manu" )
   END_RUNG wire#w1
   RUNG wire#w1
      R_Coil( "M17.3" )
   END_RUNG
   RUNG wire#w1
      R_Coil( "M16.2" )
   END_RUNG
   // the same network as SCL:
   IF ("M17.3" AND "Auto" AND "DB09_TablePos".Req1_Pos AND NOT "Timer".T10.Q AND "E16") OR ("M16.2" AND NOT "DB04_Conveyor".dbx4_0 AND NOT "TransitIn" AND NOT "TransitOut" AND "Manu") THEN
       "M16.0" := TRUE;
   END_IF;
   #_w1 := ("M17.3" AND "Auto" AND "DB09_TablePos".Req1_Pos AND NOT "Timer".T10.Q AND "E16") OR ("M16.2" AND NOT "DB04_Conveyor".dbx4_0 AND NOT "TransitIn" AND NOT "TransitOut" AND "Manu");
   IF #_w1 THEN
       "M17.3" := FALSE;
       "M16.2" := FALSE;
   END_IF;
END_REGION

REGION Network 30: Conveyor forward
   RUNG wire#powerrail
      Contact( "M16.1" )
      Contact( "E43" )
      wire#w1
      Contact( "E44" )
      wire#w2
      Contact( "Auto" )
      wire#w4
      I_Contact( "A11" )
      Coil( "ConvOk4" )
   END_RUNG
   RUNG wire#w1
      Contact( "E40" )
   END_RUNG wire#w2
   RUNG wire#w1
      I_Contact( "DB09_TablePos".dbx1_6 )
   END_RUNG wire#w2
   RUNG wire#w1
      I_Contact( "DB21_DisplayGeneralData".dbx0_2 )
   END_RUNG wire#w2
   RUNG wire#powerrail
      Contact( "M16.4" )
      Contact( "E43" )
      wire#w3
      I_Contact( "DB21_DisplayGeneralData".dbx0_5 )
      Contact( "E44" )
   END_RUNG wire#w2
   RUNG wire#powerrail
      Contact( "M16.5" )
   END_RUNG wire#w3
   RUNG wire#powerrail
      Contact( "M16.3" )
   END_RUNG wire#w3
   RUNG wire#powerrail
      Contact( "DB22_DisplayData".dbx20_1 )
      Contact( "E44" )
      I_Contact( "DB21_DisplayGeneralData".dbx0_5 )
      wire#w5
      Contact( "Manu" )
   END_RUNG wire#w4
   RUNG wire#powerrail
      Contact( "DB22_DisplayData".dbx20_0 )
      wire#w6
      Contact( "E43" )
      wire#w7
      Contact( "E40" )
      wire#w8
      I_Contact( "TransitOut" )
      I_Contact( "DB04_Conveyor".dbx4_0 )
   END_RUNG wire#w5
   RUNG wire#w6
      I_Contact( "TransitIn" )
   END_RUNG wire#w7
   RUNG wire#w7
      I_Contact( "DB09_TablePos".dbx1_6 )
   END_RUNG wire#w8
   RUNG wire#w7
      I_Contact( "DB21_DisplayGeneralData".dbx0_2 )
   END_RUNG wire#w8
   RUNG wire#w7
      I_Contact( "DB21_DisplayGeneralData".dbx0_5 )
      Contact( "DB21_DisplayGeneralData".dbx0_2 )
      Contact( "E44" )
      wire#w9
      Contact( "TransitOut" )
   END_RUNG wire#w5
   RUNG wire#w9
      I_Contact( "E40" )
   END_RUNG wire#w5
   RUNG wire#w9
      I_Contact( "DB09_TablePos".dbx1_6 )
   END_RUNG wire#w5
   RUNG wire#powerrail
      Contact( "DB22_DisplayData".dbx15_5 )
   END_RUNG wire#w5
   RUNG wire#powerrail
      Contact( "ClampCutOk19" )
   END_RUNG wire#w4
   // the same network as SCL:
   "ConvOk4" := (((("M16.1" AND "E43" AND ("E44" OR "E40" OR NOT "DB09_TablePos".dbx1_6 OR NOT "DB21_DisplayGeneralData".dbx0_2)) OR ((("M16.4" AND "E43") OR "M16.5" OR "M16.3") AND NOT "DB21_DisplayGeneralData".dbx0_5 AND "E44")) AND "Auto") OR ((("DB22_DisplayData".dbx20_1 AND "E44" AND NOT "DB21_DisplayGeneralData".dbx0_5) OR ("DB22_DisplayData".dbx20_0 AND ("E43" OR NOT "TransitIn") AND ((("E40" OR NOT "DB09_TablePos".dbx1_6 OR NOT "DB21_DisplayGeneralData".dbx0_2) AND NOT "TransitOut" AND NOT "DB04_Conveyor".dbx4_0) OR (NOT "DB21_DisplayGeneralData".dbx0_5 AND "DB21_DisplayGeneralData".dbx0_2 AND "E44" AND ("TransitOut" OR NOT "E40" OR NOT "DB09_TablePos".dbx1_6)))) OR "DB22_DisplayData".dbx15_5) AND "Manu") OR "ClampCutOk19") AND NOT "A11";
END_REGION

REGION Network 31: ConvOk7: Backward for inverter
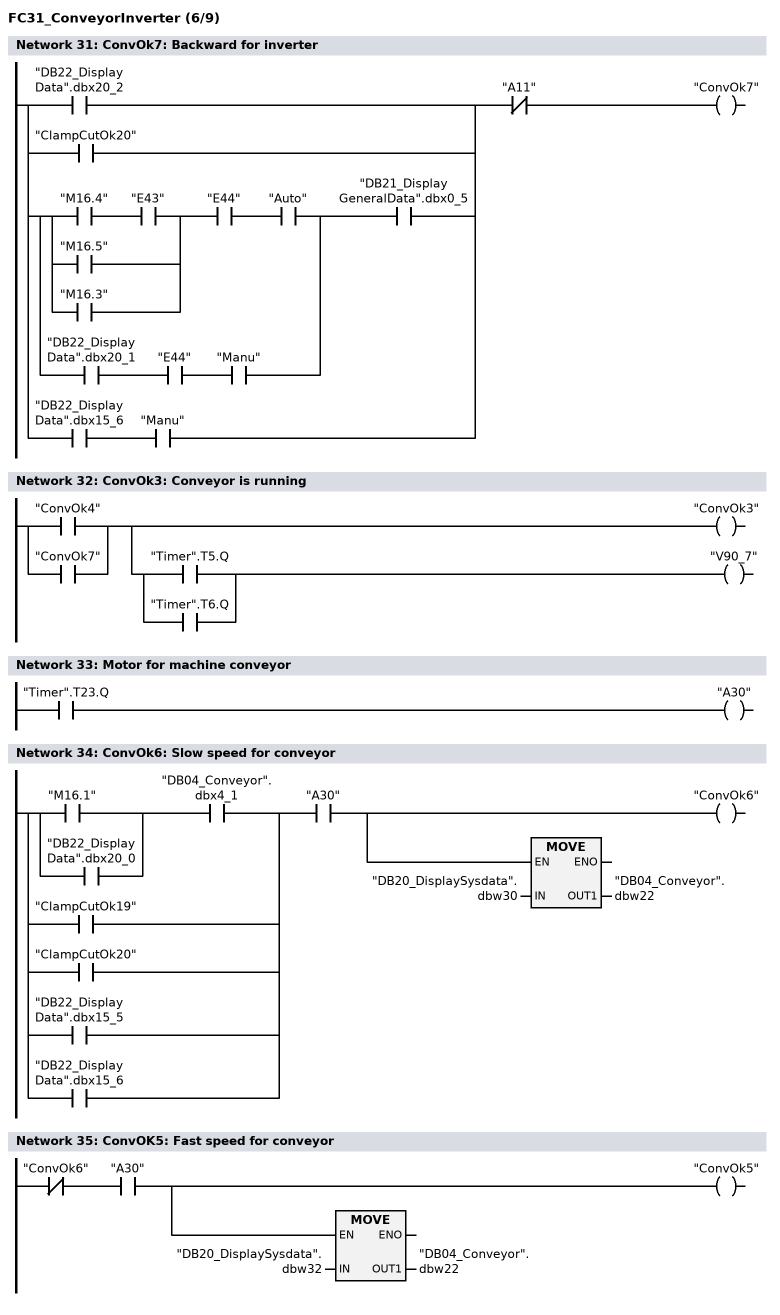
   RUNG wire#powerrail
      Contact( "DB22_DisplayData".dbx20_2 )
      wire#w1
      I_Contact( "A11" )
      Coil( "ConvOk7" )
   END_RUNG
   RUNG wire#powerrail
      Contact( "ClampCutOk20" )
   END_RUNG wire#w1
   RUNG wire#powerrail
      Contact( "M16.4" )
      Contact( "E43" )
      wire#w2
      Contact( "E44" )
      Contact( "Auto" )
      wire#w3
      Contact( "DB21_DisplayGeneralData".dbx0_5 )
   END_RUNG wire#w1
   RUNG wire#powerrail
      Contact( "M16.5" )
   END_RUNG wire#w2
   RUNG wire#powerrail
      Contact( "M16.3" )
   END_RUNG wire#w2
   RUNG wire#powerrail
      Contact( "DB22_DisplayData".dbx20_1 )
      Contact( "E44" )
      Contact( "Manu" )
   END_RUNG wire#w3
   RUNG wire#powerrail
      Contact( "DB22_DisplayData".dbx15_6 )
      Contact( "Manu" )
   END_RUNG wire#w1
   // the same network as SCL:
   "ConvOk7" := ("DB22_DisplayData".dbx20_2 OR "ClampCutOk20" OR ((((("M16.4" AND "E43") OR "M16.5" OR "M16.3") AND "E44" AND "Auto") OR ("DB22_DisplayData".dbx20_1 AND "E44" AND "Manu")) AND "DB21_DisplayGeneralData".dbx0_5) OR ("DB22_DisplayData".dbx15_6 AND "Manu")) AND NOT "A11";
END_REGION

REGION Network 32: ConvOk3: Conveyor is running
   RUNG wire#powerrail
      Contact( "ConvOk4" )
      wire#w1
      Coil( "ConvOk3" )
   END_RUNG
   RUNG wire#powerrail
      Contact( "ConvOk7" )
   END_RUNG wire#w1
   RUNG wire#w1
      Contact( "Timer".T5.Q )
      wire#w2
      Coil( "V90_7" )
   END_RUNG
   RUNG wire#w1
      Contact( "Timer".T6.Q )
   END_RUNG wire#w2
   // the same network as SCL:
   "ConvOk3" := "ConvOk4" OR "ConvOk7";
   "V90_7" := "ConvOk3" AND ("Timer".T5.Q OR "Timer".T6.Q);
END_REGION

REGION Network 33: Motor for machine conveyor
   RUNG wire#powerrail
      Contact( "Timer".T23.Q )
      Coil( "A30" )
   END_RUNG
   // the same network as SCL:
   "A30" := "Timer".T23.Q;
END_REGION

REGION Network 34: ConvOk6: Slow speed for conveyor
   RUNG wire#powerrail
      Contact( "M16.1" )
      wire#w1
      Contact( "DB04_Conveyor".dbx4_1 )
      wire#w2
      Contact( "A30" )
      wire#w3
      Coil( "ConvOk6" )
   END_RUNG
   RUNG wire#powerrail
      Contact( "DB22_DisplayData".dbx20_0 )
   END_RUNG wire#w1
   RUNG wire#powerrail
      Contact( "ClampCutOk19" )
   END_RUNG wire#w2
   RUNG wire#powerrail
      Contact( "ClampCutOk20" )
   END_RUNG wire#w2
   RUNG wire#powerrail
      Contact( "DB22_DisplayData".dbx15_5 )
   END_RUNG wire#w2
   RUNG wire#powerrail
      Contact( "DB22_DisplayData".dbx15_6 )
   END_RUNG wire#w2
   RUNG wire#w3
      { S7_GenerateENO := "TRUE" } Move(in := "DB20_DisplaySysdata".dbw30, out1 => "DB04_Conveyor".dbw22)
   END_RUNG
   // the same network as SCL:
   "ConvOk6" := ((("M16.1" OR "DB22_DisplayData".dbx20_0) AND "DB04_Conveyor".dbx4_1) OR "ClampCutOk19" OR "ClampCutOk20" OR "DB22_DisplayData".dbx15_5 OR "DB22_DisplayData".dbx15_6) AND "A30";
   IF "ConvOk6" THEN "DB04_Conveyor".dbw22 := "DB20_DisplaySysdata".dbw30; END_IF;
END_REGION

REGION Network 35: ConvOK5: Fast speed for conveyor
   RUNG wire#powerrail
      I_Contact( "ConvOk6" )
      Contact( "A30" )
      wire#w1
      Coil( "ConvOk5" )
   END_RUNG
   RUNG wire#w1
      { S7_GenerateENO := "TRUE" } Move(in := "DB20_DisplaySysdata".dbw32, out1 => "DB04_Conveyor".dbw22)
   END_RUNG
   // the same network as SCL:
   "ConvOk5" := NOT "ConvOk6" AND "A30";
   IF "ConvOk5" THEN "DB04_Conveyor".dbw22 := "DB20_DisplaySysdata".dbw32; END_IF;
END_REGION

REGION Network 36: rotation inverter: Support for speed selection
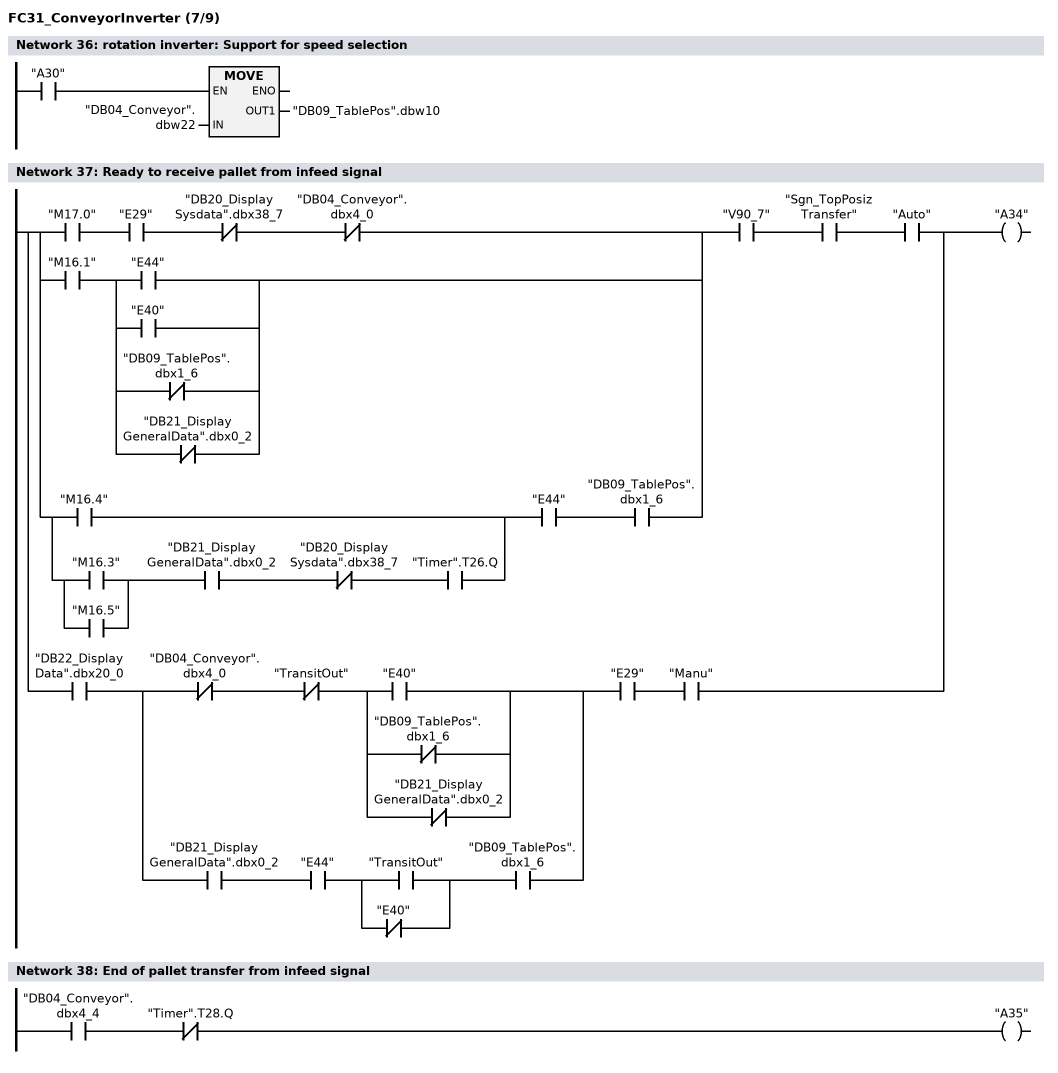
   RUNG wire#powerrail
      Contact( "A30" )
      { S7_GenerateENO := "TRUE" } Move(in := "DB04_Conveyor".dbw22, out1 => "DB09_TablePos".dbw10)
   END_RUNG
   // the same network as SCL:
   IF "A30" THEN "DB09_TablePos".dbw10 := "DB04_Conveyor".dbw22; END_IF;
END_REGION

REGION Network 37: Ready to receive pallet from infeed signal
   RUNG wire#powerrail
      Contact( "M17.0" )
      Contact( "E29" )
      I_Contact( "DB20_DisplaySysdata".dbx38_7 )
      I_Contact( "DB04_Conveyor".dbx4_0 )
      wire#w1
      Contact( "V90_7" )
      Contact( "Sgn_TopPosizTransfer" )
      Contact( "Auto" )
      wire#w5
      Coil( "A34" )
   END_RUNG
   RUNG wire#powerrail
      Contact( "M16.1" )
      wire#w2
      Contact( "E44" )
   END_RUNG wire#w1
   RUNG wire#w2
      Contact( "E40" )
   END_RUNG wire#w1
   RUNG wire#w2
      I_Contact( "DB09_TablePos".dbx1_6 )
   END_RUNG wire#w1
   RUNG wire#w2
      I_Contact( "DB21_DisplayGeneralData".dbx0_2 )
   END_RUNG wire#w1
   RUNG wire#powerrail
      Contact( "M16.4" )
      wire#w3
      Contact( "E44" )
      Contact( "DB09_TablePos".dbx1_6 )
   END_RUNG wire#w1
   RUNG wire#powerrail
      Contact( "M16.3" )
      wire#w4
      Contact( "DB21_DisplayGeneralData".dbx0_2 )
      I_Contact( "DB20_DisplaySysdata".dbx38_7 )
      Contact( "Timer".T26.Q )
   END_RUNG wire#w3
   RUNG wire#powerrail
      Contact( "M16.5" )
   END_RUNG wire#w4
   RUNG wire#powerrail
      Contact( "DB22_DisplayData".dbx20_0 )
      wire#w6
      I_Contact( "DB04_Conveyor".dbx4_0 )
      I_Contact( "TransitOut" )
      wire#w7
      Contact( "E40" )
      wire#w8
      Contact( "E29" )
      Contact( "Manu" )
   END_RUNG wire#w5
   RUNG wire#w7
      I_Contact( "DB09_TablePos".dbx1_6 )
   END_RUNG wire#w8
   RUNG wire#w7
      I_Contact( "DB21_DisplayGeneralData".dbx0_2 )
   END_RUNG wire#w8
   RUNG wire#w6
      Contact( "DB21_DisplayGeneralData".dbx0_2 )
      Contact( "E44" )
      wire#w9
      Contact( "TransitOut" )
      wire#w10
      Contact( "DB09_TablePos".dbx1_6 )
   END_RUNG wire#w8
   RUNG wire#w9
      I_Contact( "E40" )
   END_RUNG wire#w10
   // the same network as SCL:
   "A34" := ((("M17.0" AND "E29" AND NOT "DB20_DisplaySysdata".dbx38_7 AND NOT "DB04_Conveyor".dbx4_0) OR ("M16.1" AND ("E44" OR "E40" OR NOT "DB09_TablePos".dbx1_6 OR NOT "DB21_DisplayGeneralData".dbx0_2)) OR (("M16.4" OR (("M16.3" OR "M16.5") AND "DB21_DisplayGeneralData".dbx0_2 AND NOT "DB20_DisplaySysdata".dbx38_7 AND "Timer".T26.Q)) AND "E44" AND "DB09_TablePos".dbx1_6)) AND "V90_7" AND "Sgn_TopPosizTransfer" AND "Auto") OR ("DB22_DisplayData".dbx20_0 AND ((NOT "DB04_Conveyor".dbx4_0 AND NOT "TransitOut" AND ("E40" OR NOT "DB09_TablePos".dbx1_6 OR NOT "DB21_DisplayGeneralData".dbx0_2)) OR ("DB21_DisplayGeneralData".dbx0_2 AND "E44" AND ("TransitOut" OR NOT "E40") AND "DB09_TablePos".dbx1_6)) AND "E29" AND "Manu");
END_REGION

REGION Network 38: End of pallet transfer from infeed signal
   RUNG wire#powerrail
      Contact( "DB04_Conveyor".dbx4_4 )
      I_Contact( "Timer".T28.Q )
      Coil( "A35" )
   END_RUNG
   // the same network as SCL:
   "A35" := "DB04_Conveyor".dbx4_4 AND NOT "Timer".T28.Q;
END_REGION

REGION Network 39: Pallet ready for outfeed signal
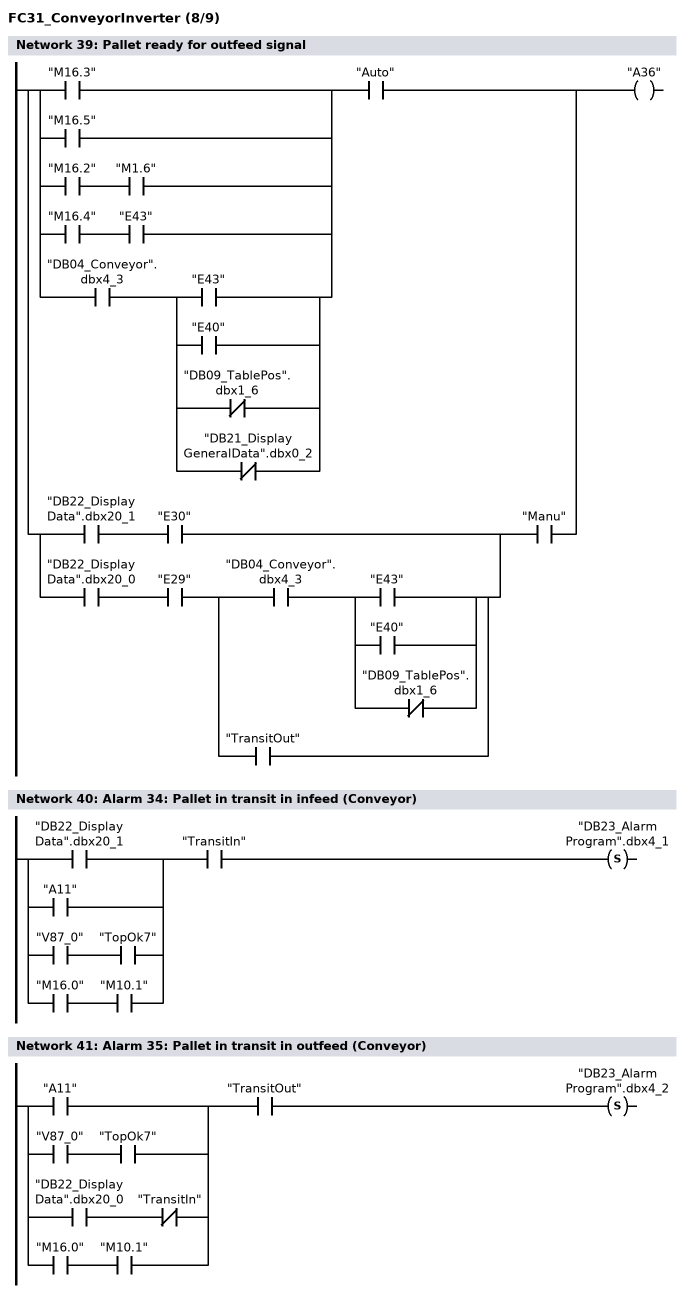
   RUNG wire#powerrail
      Contact( "M16.3" )
      wire#w1
      Contact( "Auto" )
      wire#w3
      Coil( "A36" )
   END_RUNG
   RUNG wire#powerrail
      Contact( "M16.5" )
   END_RUNG wire#w1
   RUNG wire#powerrail
      Contact( "M16.2" )
      Contact( "M1.6" )
   END_RUNG wire#w1
   RUNG wire#powerrail
      Contact( "M16.4" )
      Contact( "E43" )
   END_RUNG wire#w1
   RUNG wire#powerrail
      Contact( "DB04_Conveyor".dbx4_3 )
      wire#w2
      Contact( "E43" )
   END_RUNG wire#w1
   RUNG wire#w2
      Contact( "E40" )
   END_RUNG wire#w1
   RUNG wire#w2
      I_Contact( "DB09_TablePos".dbx1_6 )
   END_RUNG wire#w1
   RUNG wire#w2
      I_Contact( "DB21_DisplayGeneralData".dbx0_2 )
   END_RUNG wire#w1
   RUNG wire#powerrail
      Contact( "DB22_DisplayData".dbx20_1 )
      Contact( "E30" )
      wire#w4
      Contact( "Manu" )
   END_RUNG wire#w3
   RUNG wire#powerrail
      Contact( "DB22_DisplayData".dbx20_0 )
      Contact( "E29" )
      wire#w5
      Contact( "DB04_Conveyor".dbx4_3 )
      wire#w6
      Contact( "E43" )
   END_RUNG wire#w4
   RUNG wire#w6
      Contact( "E40" )
   END_RUNG wire#w4
   RUNG wire#w6
      I_Contact( "DB09_TablePos".dbx1_6 )
   END_RUNG wire#w4
   RUNG wire#w5
      Contact( "TransitOut" )
   END_RUNG wire#w4
   // the same network as SCL:
   "A36" := (("M16.3" OR "M16.5" OR ("M16.2" AND "M1.6") OR ("M16.4" AND "E43") OR ("DB04_Conveyor".dbx4_3 AND ("E43" OR "E40" OR NOT "DB09_TablePos".dbx1_6 OR NOT "DB21_DisplayGeneralData".dbx0_2))) AND "Auto") OR ((("DB22_DisplayData".dbx20_1 AND "E30") OR ("DB22_DisplayData".dbx20_0 AND "E29" AND (("DB04_Conveyor".dbx4_3 AND ("E43" OR "E40" OR NOT "DB09_TablePos".dbx1_6)) OR "TransitOut"))) AND "Manu");
END_REGION

REGION Network 40: Alarm 34: Pallet in transit in infeed (Conveyor)
   RUNG wire#powerrail
      Contact( "DB22_DisplayData".dbx20_1 )
      wire#w1
      Contact( "TransitIn" )
      S_Coil( "DB23_AlarmProgram".dbx4_1 )
   END_RUNG
   RUNG wire#powerrail
      Contact( "A11" )
   END_RUNG wire#w1
   RUNG wire#powerrail
      Contact( "V87_0" )
      Contact( "TopOk7" )
   END_RUNG wire#w1
   RUNG wire#powerrail
      Contact( "M16.0" )
      Contact( "M10.1" )
   END_RUNG wire#w1
   // the same network as SCL:
   IF ("DB22_DisplayData".dbx20_1 OR "A11" OR ("V87_0" AND "TopOk7") OR ("M16.0" AND "M10.1")) AND "TransitIn" THEN
       "DB23_AlarmProgram".dbx4_1 := TRUE;
   END_IF;
END_REGION

REGION Network 41: Alarm 35: Pallet in transit in outfeed (Conveyor)
   RUNG wire#powerrail
      Contact( "A11" )
      wire#w1
      Contact( "TransitOut" )
      S_Coil( "DB23_AlarmProgram".dbx4_2 )
   END_RUNG
   RUNG wire#powerrail
      Contact( "V87_0" )
      Contact( "TopOk7" )
   END_RUNG wire#w1
   RUNG wire#powerrail
      Contact( "DB22_DisplayData".dbx20_0 )
      I_Contact( "TransitIn" )
   END_RUNG wire#w1
   RUNG wire#powerrail
      Contact( "M16.0" )
      Contact( "M10.1" )
   END_RUNG wire#w1
   // the same network as SCL:
   IF ("A11" OR ("V87_0" AND "TopOk7") OR ("DB22_DisplayData".dbx20_0 AND NOT "TransitIn") OR ("M16.0" AND "M10.1")) AND "TransitOut" THEN
       "DB23_AlarmProgram".dbx4_2 := TRUE;
   END_IF;
END_REGION

REGION Network 42: Alarm 39: Technoplat table not in load phase
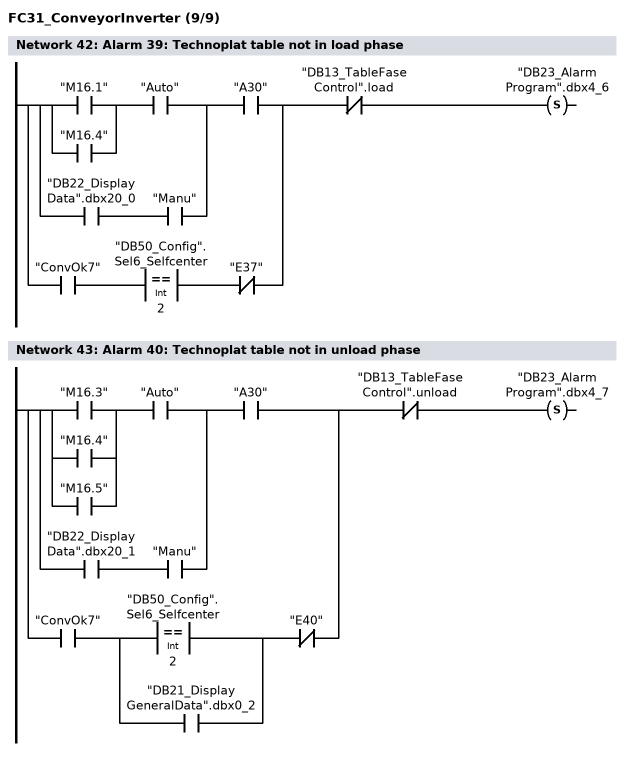
   RUNG wire#powerrail
      Contact( "M16.1" )
      wire#w1
      Contact( "Auto" )
      wire#w2
      Contact( "A30" )
      wire#w3
      I_Contact( "DB13_TableFaseControl".load )
      S_Coil( "DB23_AlarmProgram".dbx4_6 )
   END_RUNG
   RUNG wire#powerrail
      Contact( "M16.4" )
   END_RUNG wire#w1
   RUNG wire#powerrail
      Contact( "DB22_DisplayData".dbx20_0 )
      Contact( "Manu" )
   END_RUNG wire#w2
   RUNG wire#powerrail
      Contact( "ConvOk7" )
      { S7_Templates := "SrcType := Int" } EQ_Contact(in1 := "DB50_Config".Sel6_Selfcenter, in2 := 2)
      I_Contact( "E37" )
   END_RUNG wire#w3
   // the same network as SCL:
   IF ((((("M16.1" OR "M16.4") AND "Auto") OR ("DB22_DisplayData".dbx20_0 AND "Manu")) AND "A30") OR ("ConvOk7" AND ("DB50_Config".Sel6_Selfcenter = 2) AND NOT "E37")) AND NOT "DB13_TableFaseControl".load THEN
       "DB23_AlarmProgram".dbx4_6 := TRUE;
   END_IF;
END_REGION

REGION Network 43: Alarm 40: Technoplat table not in unload phase
   RUNG wire#powerrail
      Contact( "M16.3" )
      wire#w1
      Contact( "Auto" )
      wire#w2
      Contact( "A30" )
      wire#w3
      I_Contact( "DB13_TableFaseControl".unload )
      S_Coil( "DB23_AlarmProgram".dbx4_7 )
   END_RUNG
   RUNG wire#powerrail
      Contact( "M16.4" )
   END_RUNG wire#w1
   RUNG wire#powerrail
      Contact( "M16.5" )
   END_RUNG wire#w1
   RUNG wire#powerrail
      Contact( "DB22_DisplayData".dbx20_1 )
      Contact( "Manu" )
   END_RUNG wire#w2
   RUNG wire#powerrail
      Contact( "ConvOk7" )
      wire#w4
      { S7_Templates := "SrcType := Int" } EQ_Contact(in1 := "DB50_Config".Sel6_Selfcenter, in2 := 2)
      wire#w5
      I_Contact( "E40" )
   END_RUNG wire#w3
   RUNG wire#w4
      Contact( "DB21_DisplayGeneralData".dbx0_2 )
   END_RUNG wire#w5
   // the same network as SCL:
   IF ((((("M16.3" OR "M16.4" OR "M16.5") AND "Auto") OR ("DB22_DisplayData".dbx20_1 AND "Manu")) AND "A30") OR ("ConvOk7" AND (("DB50_Config".Sel6_Selfcenter = 2) OR "DB21_DisplayGeneralData".dbx0_2) AND NOT "E40")) AND NOT "DB13_TableFaseControl".unload THEN
       "DB23_AlarmProgram".dbx4_7 := TRUE;
   END_IF;
END_REGION
END_FUNCTION

FUNCTION "FC86_Conveyor_5_IN_3_OUT" : Void   // FC86, LAD
TITLE = Conveyor_5_IN_3_OUT
{ S7_Optimized_Access := 'TRUE' }
VERSION : 0.1
// 5+3 (Fitembal)
// stored: AutoNumber false, IsIECCheckEnabled false, SetENOAutomatically false, UDAEnableTagReadback false
   VAR_TEMP   // added for the SCL form of the ladder/FBD networks
      _w1 : Bool;
      _w2 : Bool;
   END_VAR
BEGIN

REGION Network 1: Manual operation for conveyor
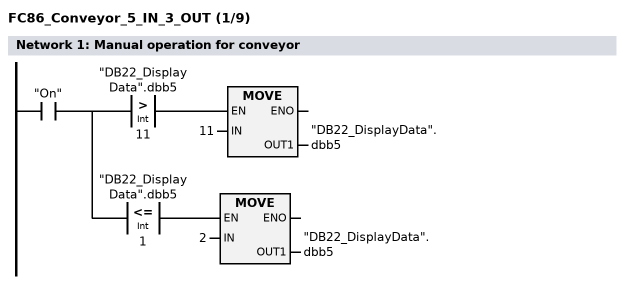
   RUNG wire#powerrail
      Contact( "On" )
      wire#w1
      { S7_Templates := "SrcType := Int" } GT_Contact(in1 := "DB22_DisplayData".dbb5, in2 := 11)
      { S7_GenerateENO := "TRUE" } Move(in := 11, out1 => "DB22_DisplayData".dbb5)
   END_RUNG
   RUNG wire#w1
      { S7_Templates := "SrcType := Int" } LE_Contact(in1 := "DB22_DisplayData".dbb5, in2 := 1)
      { S7_GenerateENO := "TRUE" } Move(in := 2, out1 => "DB22_DisplayData".dbb5)
   END_RUNG
   // the same network as SCL:
   IF "On" AND ("DB22_DisplayData".dbb5 > 11) THEN "DB22_DisplayData".dbb5 := 11; END_IF;
   IF "On" AND ("DB22_DisplayData".dbb5 <= 1) THEN "DB22_DisplayData".dbb5 := 2; END_IF;
END_REGION

REGION Network 2: Manual operation for conveyor
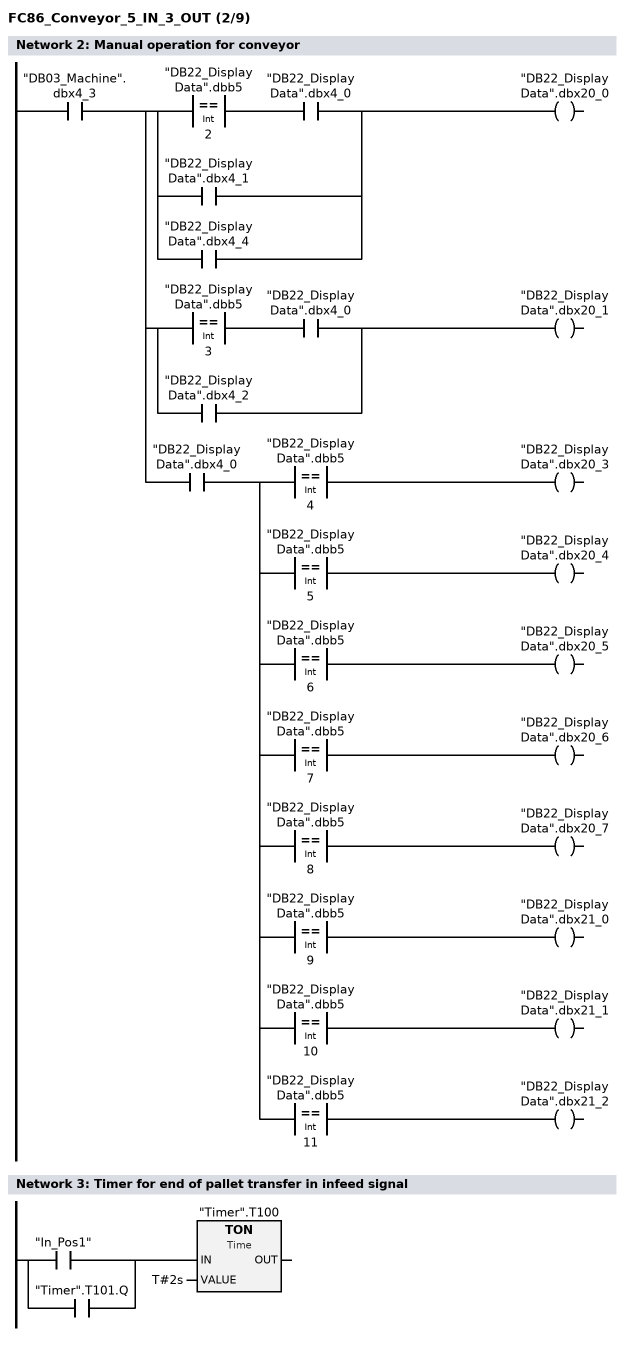
   RUNG wire#powerrail
      Contact( "DB03_Machine".dbx4_3 )
      wire#w1
      { S7_Templates := "SrcType := Int" } EQ_Contact(in1 := "DB22_DisplayData".dbb5, in2 := 2)
      Contact( "DB22_DisplayData".dbx4_0 )
      wire#w2
      Coil( "DB22_DisplayData".dbx20_0 )
   END_RUNG
   RUNG wire#w1
      Contact( "DB22_DisplayData".dbx4_1 )
   END_RUNG wire#w2
   RUNG wire#w1
      Contact( "DB22_DisplayData".dbx4_4 )
   END_RUNG wire#w2
   RUNG wire#w1
      { S7_Templates := "SrcType := Int" } EQ_Contact(in1 := "DB22_DisplayData".dbb5, in2 := 3)
      Contact( "DB22_DisplayData".dbx4_0 )
      wire#w3
      Coil( "DB22_DisplayData".dbx20_1 )
   END_RUNG
   RUNG wire#w1
      Contact( "DB22_DisplayData".dbx4_2 )
   END_RUNG wire#w3
   RUNG wire#w1
      Contact( "DB22_DisplayData".dbx4_0 )
      wire#w4
      { S7_Templates := "SrcType := Int" } EQ_Contact(in1 := "DB22_DisplayData".dbb5, in2 := 4)
      Coil( "DB22_DisplayData".dbx20_3 )
   END_RUNG
   RUNG wire#w4
      { S7_Templates := "SrcType := Int" } EQ_Contact(in1 := "DB22_DisplayData".dbb5, in2 := 5)
      Coil( "DB22_DisplayData".dbx20_4 )
   END_RUNG
   RUNG wire#w4
      { S7_Templates := "SrcType := Int" } EQ_Contact(in1 := "DB22_DisplayData".dbb5, in2 := 6)
      Coil( "DB22_DisplayData".dbx20_5 )
   END_RUNG
   RUNG wire#w4
      { S7_Templates := "SrcType := Int" } EQ_Contact(in1 := "DB22_DisplayData".dbb5, in2 := 7)
      Coil( "DB22_DisplayData".dbx20_6 )
   END_RUNG
   RUNG wire#w4
      { S7_Templates := "SrcType := Int" } EQ_Contact(in1 := "DB22_DisplayData".dbb5, in2 := 8)
      Coil( "DB22_DisplayData".dbx20_7 )
   END_RUNG
   RUNG wire#w4
      { S7_Templates := "SrcType := Int" } EQ_Contact(in1 := "DB22_DisplayData".dbb5, in2 := 9)
      Coil( "DB22_DisplayData".dbx21_0 )
   END_RUNG
   RUNG wire#w4
      { S7_Templates := "SrcType := Int" } EQ_Contact(in1 := "DB22_DisplayData".dbb5, in2 := 10)
      Coil( "DB22_DisplayData".dbx21_1 )
   END_RUNG
   RUNG wire#w4
      { S7_Templates := "SrcType := Int" } EQ_Contact(in1 := "DB22_DisplayData".dbb5, in2 := 11)
      Coil( "DB22_DisplayData".dbx21_2 )
   END_RUNG
   // the same network as SCL:
   "DB22_DisplayData".dbx20_0 := "DB03_Machine".dbx4_3 AND ((("DB22_DisplayData".dbb5 = 2) AND "DB22_DisplayData".dbx4_0) OR "DB22_DisplayData".dbx4_1 OR "DB22_DisplayData".dbx4_4);
   "DB22_DisplayData".dbx20_1 := "DB03_Machine".dbx4_3 AND ((("DB22_DisplayData".dbb5 = 3) AND "DB22_DisplayData".dbx4_0) OR "DB22_DisplayData".dbx4_2);
   #_w1 := "DB03_Machine".dbx4_3 AND "DB22_DisplayData".dbx4_0;
   "DB22_DisplayData".dbx20_3 := #_w1 AND ("DB22_DisplayData".dbb5 = 4);
   "DB22_DisplayData".dbx20_4 := #_w1 AND ("DB22_DisplayData".dbb5 = 5);
   "DB22_DisplayData".dbx20_5 := #_w1 AND ("DB22_DisplayData".dbb5 = 6);
   "DB22_DisplayData".dbx20_6 := #_w1 AND ("DB22_DisplayData".dbb5 = 7);
   "DB22_DisplayData".dbx20_7 := #_w1 AND ("DB22_DisplayData".dbb5 = 8);
   "DB22_DisplayData".dbx21_0 := #_w1 AND ("DB22_DisplayData".dbb5 = 9);
   "DB22_DisplayData".dbx21_1 := #_w1 AND ("DB22_DisplayData".dbb5 = 10);
   "DB22_DisplayData".dbx21_2 := #_w1 AND ("DB22_DisplayData".dbb5 = 11);
END_REGION

REGION Network 3: Timer for end of pallet transfer in infeed signal
   "Timer".T100.TON(IN := "In_Pos1" OR "Timer".T101.Q, PT := T#2s);   // TON coil
END_REGION

REGION Network 4: Timeout for conveyor pos1
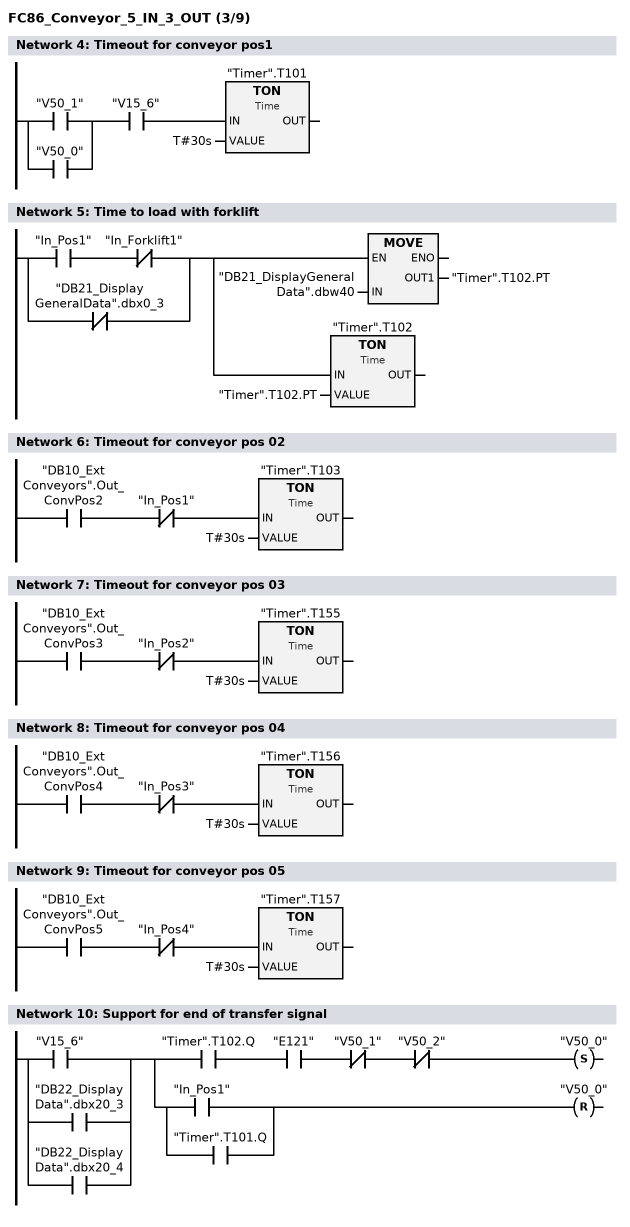
   "Timer".T101.TON(IN := ("V50_1" OR "V50_0") AND "V15_6", PT := T#30s);   // TON coil
END_REGION

REGION Network 5: Time to load with forklift
   #_w1 := ("In_Pos1" AND NOT "In_Forklift1") OR NOT "DB21_DisplayGeneralData".dbx0_3;
   IF #_w1 THEN "Timer".T102.PT := "DB21_DisplayGeneralData".dbw40; END_IF;
   "Timer".T102.TON(IN := #_w1, PT := "Timer".T102.PT);   // TON coil
END_REGION

REGION Network 6: Timeout for conveyor pos 02
   "Timer".T103.TON(IN := "DB10_ExtConveyors".Out_ConvPos2 AND NOT "In_Pos1", PT := T#30s);   // TON coil
END_REGION

REGION Network 7: Timeout for conveyor pos 03
   "Timer".T155.TON(IN := "DB10_ExtConveyors".Out_ConvPos3 AND NOT "In_Pos2", PT := T#30s);   // TON coil
END_REGION

REGION Network 8: Timeout for conveyor pos 04
   "Timer".T156.TON(IN := "DB10_ExtConveyors".Out_ConvPos4 AND NOT "In_Pos3", PT := T#30s);   // TON coil
END_REGION

REGION Network 9: Timeout for conveyor pos 05
   "Timer".T157.TON(IN := "DB10_ExtConveyors".Out_ConvPos5 AND NOT "In_Pos4", PT := T#30s);   // TON coil
END_REGION

REGION Network 10: Support for end of transfer signal
   RUNG wire#powerrail
      Contact( "V15_6" )
      wire#w1
      Contact( "Timer".T102.Q )
      Contact( "E121" )
      I_Contact( "V50_1" )
      I_Contact( "V50_2" )
      S_Coil( "V50_0" )
   END_RUNG
   RUNG wire#powerrail
      Contact( "DB22_DisplayData".dbx20_3 )
   END_RUNG wire#w1
   RUNG wire#powerrail
      Contact( "DB22_DisplayData".dbx20_4 )
   END_RUNG wire#w1
   RUNG wire#w1
      Contact( "In_Pos1" )
      wire#w2
      R_Coil( "V50_0" )
   END_RUNG
   RUNG wire#w1
      Contact( "Timer".T101.Q )
   END_RUNG wire#w2
   // the same network as SCL:
   #_w1 := "V15_6" OR "DB22_DisplayData".dbx20_3 OR "DB22_DisplayData".dbx20_4;
   IF #_w1 AND "Timer".T102.Q AND "E121" AND NOT "V50_1" AND NOT "V50_2" THEN "V50_0" := TRUE; END_IF;
   IF #_w1 AND ("In_Pos1" OR "Timer".T101.Q) THEN "V50_0" := FALSE; END_IF;
END_REGION

REGION Network 11: Transit memory for conveyor pos1
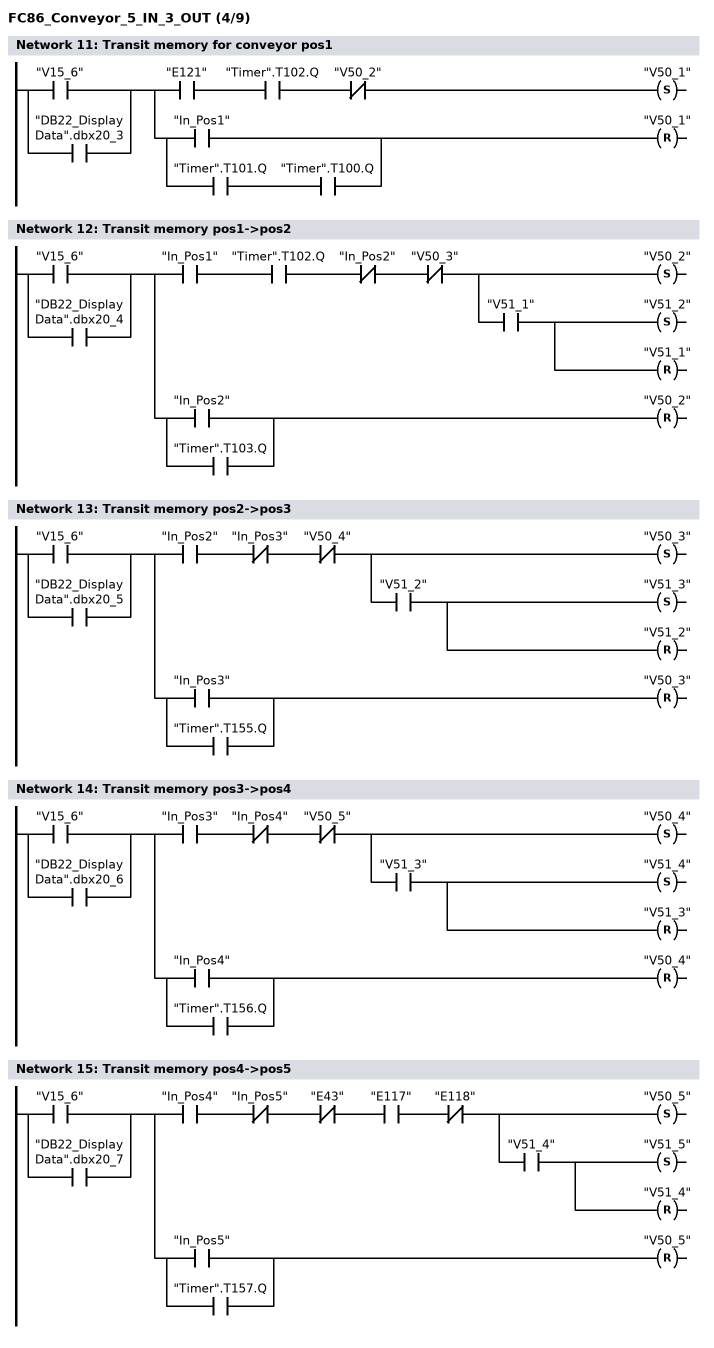
   RUNG wire#powerrail
      Contact( "V15_6" )
      wire#w1
      Contact( "E121" )
      Contact( "Timer".T102.Q )
      I_Contact( "V50_2" )
      S_Coil( "V50_1" )
   END_RUNG
   RUNG wire#powerrail
      Contact( "DB22_DisplayData".dbx20_3 )
   END_RUNG wire#w1
   RUNG wire#w1
      Contact( "In_Pos1" )
      wire#w2
      R_Coil( "V50_1" )
   END_RUNG
   RUNG wire#w1
      Contact( "Timer".T101.Q )
      Contact( "Timer".T100.Q )
   END_RUNG wire#w2
   // the same network as SCL:
   #_w1 := "V15_6" OR "DB22_DisplayData".dbx20_3;
   IF #_w1 AND "E121" AND "Timer".T102.Q AND NOT "V50_2" THEN "V50_1" := TRUE; END_IF;
   IF #_w1 AND ("In_Pos1" OR ("Timer".T101.Q AND "Timer".T100.Q)) THEN "V50_1" := FALSE; END_IF;
END_REGION

REGION Network 12: Transit memory pos1->pos2
   RUNG wire#powerrail
      Contact( "V15_6" )
      wire#w1
      Contact( "In_Pos1" )
      Contact( "Timer".T102.Q )
      I_Contact( "In_Pos2" )
      I_Contact( "V50_3" )
      wire#w2
      S_Coil( "V50_2" )
   END_RUNG
   RUNG wire#powerrail
      Contact( "DB22_DisplayData".dbx20_4 )
   END_RUNG wire#w1
   RUNG wire#w2
      Contact( "V51_1" )
      wire#w3
      S_Coil( "V51_2" )
   END_RUNG
   RUNG wire#w3
      R_Coil( "V51_1" )
   END_RUNG
   RUNG wire#w1
      Contact( "In_Pos2" )
      wire#w4
      R_Coil( "V50_2" )
   END_RUNG
   RUNG wire#w1
      Contact( "Timer".T103.Q )
   END_RUNG wire#w4
   // the same network as SCL:
   #_w1 := "V15_6" OR "DB22_DisplayData".dbx20_4;
   #_w2 := #_w1 AND "In_Pos1" AND "Timer".T102.Q AND NOT "In_Pos2" AND NOT "V50_3";
   IF #_w2 THEN "V50_2" := TRUE; END_IF;
   IF #_w2 AND "V51_1" THEN
       "V51_2" := TRUE;
       "V51_1" := FALSE;
   END_IF;
   IF #_w1 AND ("In_Pos2" OR "Timer".T103.Q) THEN "V50_2" := FALSE; END_IF;
END_REGION

REGION Network 13: Transit memory pos2->pos3
   RUNG wire#powerrail
      Contact( "V15_6" )
      wire#w1
      Contact( "In_Pos2" )
      I_Contact( "In_Pos3" )
      I_Contact( "V50_4" )
      wire#w2
      S_Coil( "V50_3" )
   END_RUNG
   RUNG wire#powerrail
      Contact( "DB22_DisplayData".dbx20_5 )
   END_RUNG wire#w1
   RUNG wire#w2
      Contact( "V51_2" )
      wire#w3
      S_Coil( "V51_3" )
   END_RUNG
   RUNG wire#w3
      R_Coil( "V51_2" )
   END_RUNG
   RUNG wire#w1
      Contact( "In_Pos3" )
      wire#w4
      R_Coil( "V50_3" )
   END_RUNG
   RUNG wire#w1
      Contact( "Timer".T155.Q )
   END_RUNG wire#w4
   // the same network as SCL:
   #_w1 := "V15_6" OR "DB22_DisplayData".dbx20_5;
   #_w2 := #_w1 AND "In_Pos2" AND NOT "In_Pos3" AND NOT "V50_4";
   IF #_w2 THEN "V50_3" := TRUE; END_IF;
   IF #_w2 AND "V51_2" THEN
       "V51_3" := TRUE;
       "V51_2" := FALSE;
   END_IF;
   IF #_w1 AND ("In_Pos3" OR "Timer".T155.Q) THEN "V50_3" := FALSE; END_IF;
END_REGION

REGION Network 14: Transit memory pos3->pos4
   RUNG wire#powerrail
      Contact( "V15_6" )
      wire#w1
      Contact( "In_Pos3" )
      I_Contact( "In_Pos4" )
      I_Contact( "V50_5" )
      wire#w2
      S_Coil( "V50_4" )
   END_RUNG
   RUNG wire#powerrail
      Contact( "DB22_DisplayData".dbx20_6 )
   END_RUNG wire#w1
   RUNG wire#w2
      Contact( "V51_3" )
      wire#w3
      S_Coil( "V51_4" )
   END_RUNG
   RUNG wire#w3
      R_Coil( "V51_3" )
   END_RUNG
   RUNG wire#w1
      Contact( "In_Pos4" )
      wire#w4
      R_Coil( "V50_4" )
   END_RUNG
   RUNG wire#w1
      Contact( "Timer".T156.Q )
   END_RUNG wire#w4
   // the same network as SCL:
   #_w1 := "V15_6" OR "DB22_DisplayData".dbx20_6;
   #_w2 := #_w1 AND "In_Pos3" AND NOT "In_Pos4" AND NOT "V50_5";
   IF #_w2 THEN "V50_4" := TRUE; END_IF;
   IF #_w2 AND "V51_3" THEN
       "V51_4" := TRUE;
       "V51_3" := FALSE;
   END_IF;
   IF #_w1 AND ("In_Pos4" OR "Timer".T156.Q) THEN "V50_4" := FALSE; END_IF;
END_REGION

REGION Network 15: Transit memory pos4->pos5
   RUNG wire#powerrail
      Contact( "V15_6" )
      wire#w1
      Contact( "In_Pos4" )
      I_Contact( "In_Pos5" )
      I_Contact( "E43" )
      Contact( "E117" )
      I_Contact( "E118" )
      wire#w2
      S_Coil( "V50_5" )
   END_RUNG
   RUNG wire#powerrail
      Contact( "DB22_DisplayData".dbx20_7 )
   END_RUNG wire#w1
   RUNG wire#w2
      Contact( "V51_4" )
      wire#w3
      S_Coil( "V51_5" )
   END_RUNG
   RUNG wire#w3
      R_Coil( "V51_4" )
   END_RUNG
   RUNG wire#w1
      Contact( "In_Pos5" )
      wire#w4
      R_Coil( "V50_5" )
   END_RUNG
   RUNG wire#w1
      Contact( "Timer".T157.Q )
   END_RUNG wire#w4
   // the same network as SCL:
   #_w1 := "V15_6" OR "DB22_DisplayData".dbx20_7;
   #_w2 := #_w1 AND "In_Pos4" AND NOT "In_Pos5" AND NOT "E43" AND "E117" AND NOT "E118";
   IF #_w2 THEN "V50_5" := TRUE; END_IF;
   IF #_w2 AND "V51_4" THEN
       "V51_5" := TRUE;
       "V51_4" := FALSE;
   END_IF;
   IF #_w1 AND ("In_Pos5" OR "Timer".T157.Q) THEN "V50_5" := FALSE; END_IF;
END_REGION

REGION Network 16: Ready to receive pallet in infeed signal
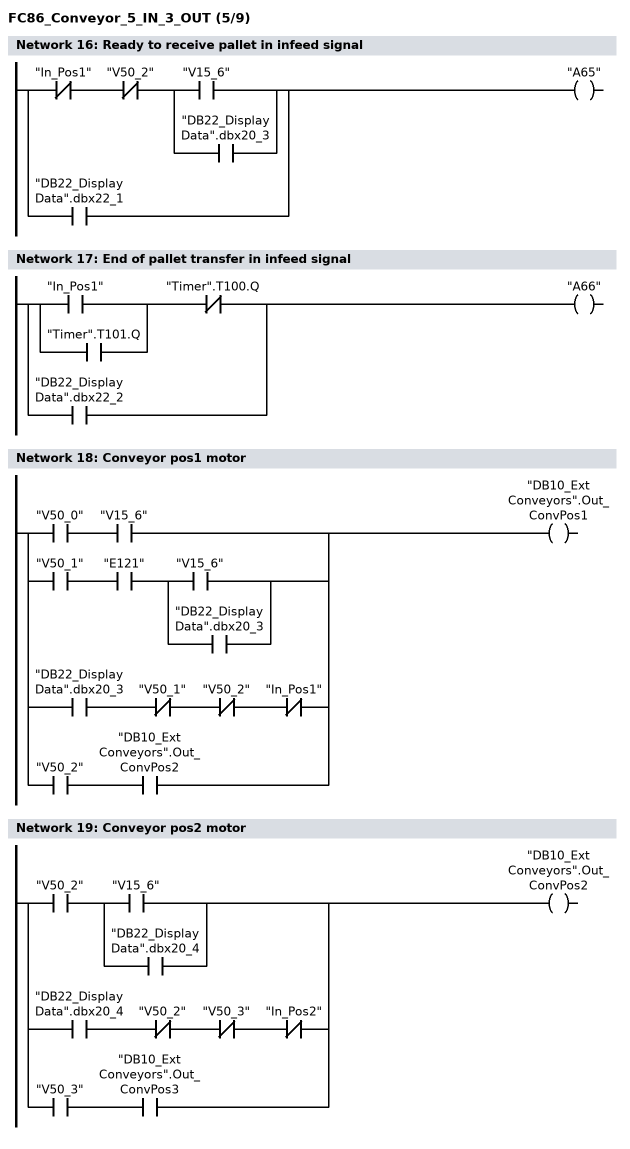
   RUNG wire#powerrail
      I_Contact( "In_Pos1" )
      I_Contact( "V50_2" )
      wire#w1
      Contact( "V15_6" )
      wire#w2
      Coil( "A65" )
   END_RUNG
   RUNG wire#w1
      Contact( "DB22_DisplayData".dbx20_3 )
   END_RUNG wire#w2
   RUNG wire#powerrail
      Contact( "DB22_DisplayData".dbx22_1 )
   END_RUNG wire#w2
   // the same network as SCL:
   "A65" := (NOT "In_Pos1" AND NOT "V50_2" AND ("V15_6" OR "DB22_DisplayData".dbx20_3)) OR "DB22_DisplayData".dbx22_1;
END_REGION

REGION Network 17: End of pallet transfer in infeed signal
   RUNG wire#powerrail
      Contact( "In_Pos1" )
      wire#w1
      I_Contact( "Timer".T100.Q )
      wire#w2
      Coil( "A66" )
   END_RUNG
   RUNG wire#powerrail
      Contact( "Timer".T101.Q )
   END_RUNG wire#w1
   RUNG wire#powerrail
      Contact( "DB22_DisplayData".dbx22_2 )
   END_RUNG wire#w2
   // the same network as SCL:
   "A66" := (("In_Pos1" OR "Timer".T101.Q) AND NOT "Timer".T100.Q) OR "DB22_DisplayData".dbx22_2;
END_REGION

REGION Network 18: Conveyor pos1 motor
   RUNG wire#powerrail
      Contact( "V50_0" )
      Contact( "V15_6" )
      wire#w1
      Coil( "DB10_ExtConveyors".Out_ConvPos1 )
   END_RUNG
   RUNG wire#powerrail
      Contact( "V50_1" )
      Contact( "E121" )
      wire#w2
      Contact( "V15_6" )
   END_RUNG wire#w1
   RUNG wire#w2
      Contact( "DB22_DisplayData".dbx20_3 )
   END_RUNG wire#w1
   RUNG wire#powerrail
      Contact( "DB22_DisplayData".dbx20_3 )
      I_Contact( "V50_1" )
      I_Contact( "V50_2" )
      I_Contact( "In_Pos1" )
   END_RUNG wire#w1
   RUNG wire#powerrail
      Contact( "V50_2" )
      Contact( "DB10_ExtConveyors".Out_ConvPos2 )
   END_RUNG wire#w1
   // the same network as SCL:
   "DB10_ExtConveyors".Out_ConvPos1 := ("V50_0" AND "V15_6") OR ("V50_1" AND "E121" AND ("V15_6" OR "DB22_DisplayData".dbx20_3)) OR ("DB22_DisplayData".dbx20_3 AND NOT "V50_1" AND NOT "V50_2" AND NOT "In_Pos1") OR ("V50_2" AND "DB10_ExtConveyors".Out_ConvPos2);
END_REGION

REGION Network 19: Conveyor pos2 motor
   RUNG wire#powerrail
      Contact( "V50_2" )
      wire#w1
      Contact( "V15_6" )
      wire#w2
      Coil( "DB10_ExtConveyors".Out_ConvPos2 )
   END_RUNG
   RUNG wire#w1
      Contact( "DB22_DisplayData".dbx20_4 )
   END_RUNG wire#w2
   RUNG wire#powerrail
      Contact( "DB22_DisplayData".dbx20_4 )
      I_Contact( "V50_2" )
      I_Contact( "V50_3" )
      I_Contact( "In_Pos2" )
   END_RUNG wire#w2
   RUNG wire#powerrail
      Contact( "V50_3" )
      Contact( "DB10_ExtConveyors".Out_ConvPos3 )
   END_RUNG wire#w2
   // the same network as SCL:
   "DB10_ExtConveyors".Out_ConvPos2 := ("V50_2" AND ("V15_6" OR "DB22_DisplayData".dbx20_4)) OR ("DB22_DisplayData".dbx20_4 AND NOT "V50_2" AND NOT "V50_3" AND NOT "In_Pos2") OR ("V50_3" AND "DB10_ExtConveyors".Out_ConvPos3);
END_REGION

REGION Network 20: Conveyor pos3 motor
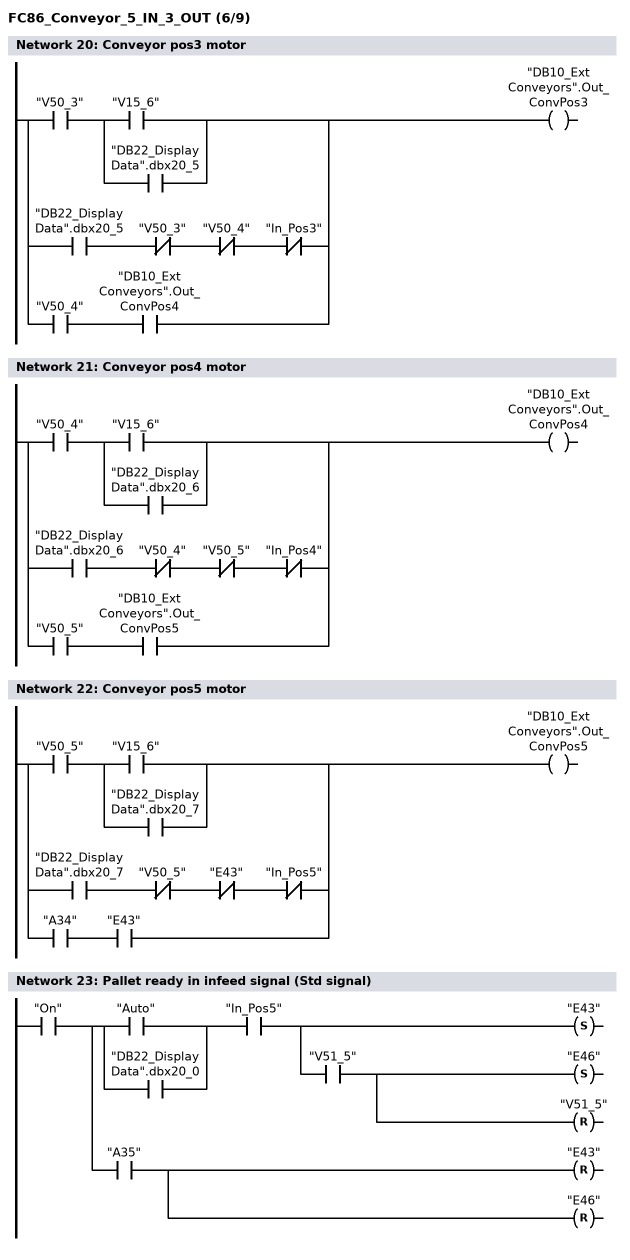
   RUNG wire#powerrail
      Contact( "V50_3" )
      wire#w1
      Contact( "V15_6" )
      wire#w2
      Coil( "DB10_ExtConveyors".Out_ConvPos3 )
   END_RUNG
   RUNG wire#w1
      Contact( "DB22_DisplayData".dbx20_5 )
   END_RUNG wire#w2
   RUNG wire#powerrail
      Contact( "DB22_DisplayData".dbx20_5 )
      I_Contact( "V50_3" )
      I_Contact( "V50_4" )
      I_Contact( "In_Pos3" )
   END_RUNG wire#w2
   RUNG wire#powerrail
      Contact( "V50_4" )
      Contact( "DB10_ExtConveyors".Out_ConvPos4 )
   END_RUNG wire#w2
   // the same network as SCL:
   "DB10_ExtConveyors".Out_ConvPos3 := ("V50_3" AND ("V15_6" OR "DB22_DisplayData".dbx20_5)) OR ("DB22_DisplayData".dbx20_5 AND NOT "V50_3" AND NOT "V50_4" AND NOT "In_Pos3") OR ("V50_4" AND "DB10_ExtConveyors".Out_ConvPos4);
END_REGION

REGION Network 21: Conveyor pos4 motor
   RUNG wire#powerrail
      Contact( "V50_4" )
      wire#w1
      Contact( "V15_6" )
      wire#w2
      Coil( "DB10_ExtConveyors".Out_ConvPos4 )
   END_RUNG
   RUNG wire#w1
      Contact( "DB22_DisplayData".dbx20_6 )
   END_RUNG wire#w2
   RUNG wire#powerrail
      Contact( "DB22_DisplayData".dbx20_6 )
      I_Contact( "V50_4" )
      I_Contact( "V50_5" )
      I_Contact( "In_Pos4" )
   END_RUNG wire#w2
   RUNG wire#powerrail
      Contact( "V50_5" )
      Contact( "DB10_ExtConveyors".Out_ConvPos5 )
   END_RUNG wire#w2
   // the same network as SCL:
   "DB10_ExtConveyors".Out_ConvPos4 := ("V50_4" AND ("V15_6" OR "DB22_DisplayData".dbx20_6)) OR ("DB22_DisplayData".dbx20_6 AND NOT "V50_4" AND NOT "V50_5" AND NOT "In_Pos4") OR ("V50_5" AND "DB10_ExtConveyors".Out_ConvPos5);
END_REGION

REGION Network 22: Conveyor pos5 motor
   RUNG wire#powerrail
      Contact( "V50_5" )
      wire#w1
      Contact( "V15_6" )
      wire#w2
      Coil( "DB10_ExtConveyors".Out_ConvPos5 )
   END_RUNG
   RUNG wire#w1
      Contact( "DB22_DisplayData".dbx20_7 )
   END_RUNG wire#w2
   RUNG wire#powerrail
      Contact( "DB22_DisplayData".dbx20_7 )
      I_Contact( "V50_5" )
      I_Contact( "E43" )
      I_Contact( "In_Pos5" )
   END_RUNG wire#w2
   RUNG wire#powerrail
      Contact( "A34" )
      Contact( "E43" )
   END_RUNG wire#w2
   // the same network as SCL:
   "DB10_ExtConveyors".Out_ConvPos5 := ("V50_5" AND ("V15_6" OR "DB22_DisplayData".dbx20_7)) OR ("DB22_DisplayData".dbx20_7 AND NOT "V50_5" AND NOT "E43" AND NOT "In_Pos5") OR ("A34" AND "E43");
END_REGION

REGION Network 23: Pallet ready in infeed signal (Std signal)
   RUNG wire#powerrail
      Contact( "On" )
      wire#w1
      Contact( "Auto" )
      wire#w2
      Contact( "In_Pos5" )
      wire#w3
      S_Coil( "E43" )
   END_RUNG
   RUNG wire#w1
      Contact( "DB22_DisplayData".dbx20_0 )
   END_RUNG wire#w2
   RUNG wire#w3
      Contact( "V51_5" )
      wire#w4
      S_Coil( "E46" )
   END_RUNG
   RUNG wire#w4
      R_Coil( "V51_5" )
   END_RUNG
   RUNG wire#w1
      Contact( "A35" )
      wire#w5
      R_Coil( "E43" )
   END_RUNG
   RUNG wire#w5
      R_Coil( "E46" )
   END_RUNG
   // the same network as SCL:
   #_w1 := "On" AND ("Auto" OR "DB22_DisplayData".dbx20_0) AND "In_Pos5";
   IF #_w1 THEN "E43" := TRUE; END_IF;
   IF #_w1 AND "V51_5" THEN
       "E46" := TRUE;
       "V51_5" := FALSE;
   END_IF;
   IF "On" AND "A35" THEN
       "E43" := FALSE;
       "E46" := FALSE;
   END_IF;
END_REGION

REGION Network 24: Memory to exclude wrapping in pos 1
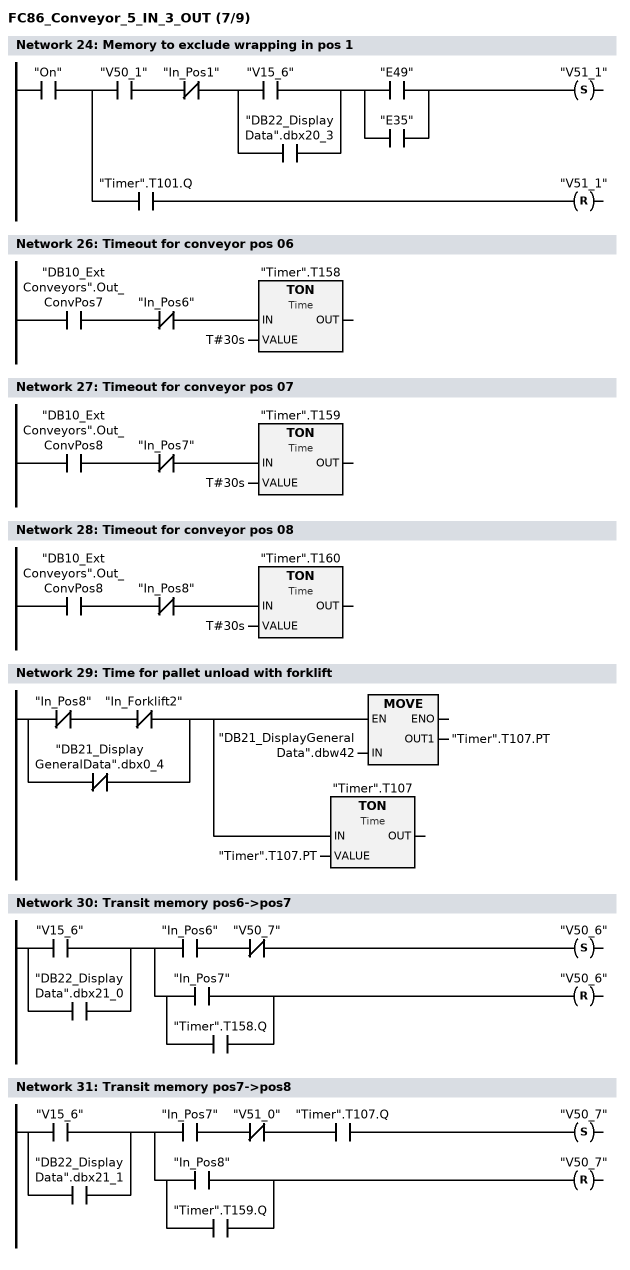
   RUNG wire#powerrail
      Contact( "On" )
      wire#w1
      Contact( "V50_1" )
      I_Contact( "In_Pos1" )
      wire#w2
      Contact( "V15_6" )
      wire#w3
      Contact( "E49" )
      wire#w4
      S_Coil( "V51_1" )
   END_RUNG
   RUNG wire#w2
      Contact( "DB22_DisplayData".dbx20_3 )
   END_RUNG wire#w3
   RUNG wire#w3
      Contact( "E35" )
   END_RUNG wire#w4
   RUNG wire#w1
      Contact( "Timer".T101.Q )
      R_Coil( "V51_1" )
   END_RUNG
   // the same network as SCL:
   IF "On" AND "V50_1" AND NOT "In_Pos1" AND ("V15_6" OR "DB22_DisplayData".dbx20_3) AND ("E49" OR "E35") THEN
       "V51_1" := TRUE;
   END_IF;
   IF "On" AND "Timer".T101.Q THEN "V51_1" := FALSE; END_IF;
END_REGION

REGION Network 25: >>>>>>> OUTFEED CONVEYOR <<<<<<<<
END_REGION

REGION Network 26: Timeout for conveyor pos 06
   "Timer".T158.TON(IN := "DB10_ExtConveyors".Out_ConvPos7 AND NOT "In_Pos6", PT := T#30s);   // TON coil
END_REGION

REGION Network 27: Timeout for conveyor pos 07
   "Timer".T159.TON(IN := "DB10_ExtConveyors".Out_ConvPos8 AND NOT "In_Pos7", PT := T#30s);   // TON coil
END_REGION

REGION Network 28: Timeout for conveyor pos 08
   "Timer".T160.TON(IN := "DB10_ExtConveyors".Out_ConvPos8 AND NOT "In_Pos8", PT := T#30s);   // TON coil
END_REGION

REGION Network 29: Time for pallet unload with forklift
   #_w1 := (NOT "In_Pos8" AND NOT "In_Forklift2") OR NOT "DB21_DisplayGeneralData".dbx0_4;
   IF #_w1 THEN "Timer".T107.PT := "DB21_DisplayGeneralData".dbw42; END_IF;
   "Timer".T107.TON(IN := #_w1, PT := "Timer".T107.PT);   // TON coil
END_REGION

REGION Network 30: Transit memory pos6->pos7
   RUNG wire#powerrail
      Contact( "V15_6" )
      wire#w1
      Contact( "In_Pos6" )
      I_Contact( "V50_7" )
      S_Coil( "V50_6" )
   END_RUNG
   RUNG wire#powerrail
      Contact( "DB22_DisplayData".dbx21_0 )
   END_RUNG wire#w1
   RUNG wire#w1
      Contact( "In_Pos7" )
      wire#w2
      R_Coil( "V50_6" )
   END_RUNG
   RUNG wire#w1
      Contact( "Timer".T158.Q )
   END_RUNG wire#w2
   // the same network as SCL:
   #_w1 := "V15_6" OR "DB22_DisplayData".dbx21_0;
   IF #_w1 AND "In_Pos6" AND NOT "V50_7" THEN "V50_6" := TRUE; END_IF;
   IF #_w1 AND ("In_Pos7" OR "Timer".T158.Q) THEN "V50_6" := FALSE; END_IF;
END_REGION

REGION Network 31: Transit memory pos7->pos8
   RUNG wire#powerrail
      Contact( "V15_6" )
      wire#w1
      Contact( "In_Pos7" )
      I_Contact( "V51_0" )
      Contact( "Timer".T107.Q )
      S_Coil( "V50_7" )
   END_RUNG
   RUNG wire#powerrail
      Contact( "DB22_DisplayData".dbx21_1 )
   END_RUNG wire#w1
   RUNG wire#w1
      Contact( "In_Pos8" )
      wire#w2
      R_Coil( "V50_7" )
   END_RUNG
   RUNG wire#w1
      Contact( "Timer".T159.Q )
   END_RUNG wire#w2
   // the same network as SCL:
   #_w1 := "V15_6" OR "DB22_DisplayData".dbx21_1;
   IF #_w1 AND "In_Pos7" AND NOT "V51_0" AND "Timer".T107.Q THEN "V50_7" := TRUE; END_IF;
   IF #_w1 AND ("In_Pos8" OR "Timer".T159.Q) THEN "V50_7" := FALSE; END_IF;
END_REGION

REGION Network 32: Outfeed conveyor pos.8 unload
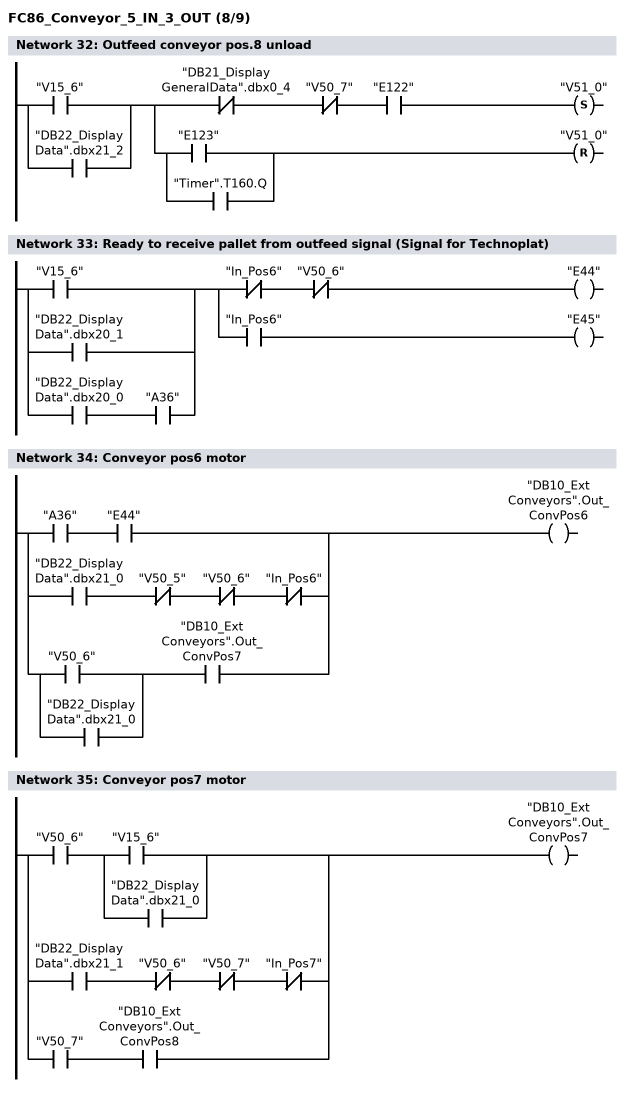
   RUNG wire#powerrail
      Contact( "V15_6" )
      wire#w1
      I_Contact( "DB21_DisplayGeneralData".dbx0_4 )
      I_Contact( "V50_7" )
      Contact( "E122" )
      S_Coil( "V51_0" )
   END_RUNG
   RUNG wire#powerrail
      Contact( "DB22_DisplayData".dbx21_2 )
   END_RUNG wire#w1
   RUNG wire#w1
      Contact( "E123" )
      wire#w2
      R_Coil( "V51_0" )
   END_RUNG
   RUNG wire#w1
      Contact( "Timer".T160.Q )
   END_RUNG wire#w2
   // the same network as SCL:
   #_w1 := "V15_6" OR "DB22_DisplayData".dbx21_2;
   IF #_w1 AND NOT "DB21_DisplayGeneralData".dbx0_4 AND NOT "V50_7" AND "E122" THEN "V51_0" := TRUE; END_IF;
   IF #_w1 AND ("E123" OR "Timer".T160.Q) THEN "V51_0" := FALSE; END_IF;
END_REGION

REGION Network 33: Ready to receive pallet from outfeed signal (Signal for Technoplat)
   RUNG wire#powerrail
      Contact( "V15_6" )
      wire#w1
      I_Contact( "In_Pos6" )
      I_Contact( "V50_6" )
      Coil( "E44" )
   END_RUNG
   RUNG wire#powerrail
      Contact( "DB22_DisplayData".dbx20_1 )
   END_RUNG wire#w1
   RUNG wire#powerrail
      Contact( "DB22_DisplayData".dbx20_0 )
      Contact( "A36" )
   END_RUNG wire#w1
   RUNG wire#w1
      Contact( "In_Pos6" )
      Coil( "E45" )
   END_RUNG
   // the same network as SCL:
   #_w1 := "V15_6" OR "DB22_DisplayData".dbx20_1 OR ("DB22_DisplayData".dbx20_0 AND "A36");
   "E44" := #_w1 AND NOT "In_Pos6" AND NOT "V50_6";
   "E45" := #_w1 AND "In_Pos6";
END_REGION

REGION Network 34: Conveyor pos6 motor
   RUNG wire#powerrail
      Contact( "A36" )
      Contact( "E44" )
      wire#w1
      Coil( "DB10_ExtConveyors".Out_ConvPos6 )
   END_RUNG
   RUNG wire#powerrail
      Contact( "DB22_DisplayData".dbx21_0 )
      I_Contact( "V50_5" )
      I_Contact( "V50_6" )
      I_Contact( "In_Pos6" )
   END_RUNG wire#w1
   RUNG wire#powerrail
      Contact( "V50_6" )
      wire#w2
      Contact( "DB10_ExtConveyors".Out_ConvPos7 )
   END_RUNG wire#w1
   RUNG wire#powerrail
      Contact( "DB22_DisplayData".dbx21_0 )
   END_RUNG wire#w2
   // the same network as SCL:
   "DB10_ExtConveyors".Out_ConvPos6 := ("A36" AND "E44") OR ("DB22_DisplayData".dbx21_0 AND NOT "V50_5" AND NOT "V50_6" AND NOT "In_Pos6") OR (("V50_6" OR "DB22_DisplayData".dbx21_0) AND "DB10_ExtConveyors".Out_ConvPos7);
END_REGION

REGION Network 35: Conveyor pos7 motor
   RUNG wire#powerrail
      Contact( "V50_6" )
      wire#w1
      Contact( "V15_6" )
      wire#w2
      Coil( "DB10_ExtConveyors".Out_ConvPos7 )
   END_RUNG
   RUNG wire#w1
      Contact( "DB22_DisplayData".dbx21_0 )
   END_RUNG wire#w2
   RUNG wire#powerrail
      Contact( "DB22_DisplayData".dbx21_1 )
      I_Contact( "V50_6" )
      I_Contact( "V50_7" )
      I_Contact( "In_Pos7" )
   END_RUNG wire#w2
   RUNG wire#powerrail
      Contact( "V50_7" )
      Contact( "DB10_ExtConveyors".Out_ConvPos8 )
   END_RUNG wire#w2
   // the same network as SCL:
   "DB10_ExtConveyors".Out_ConvPos7 := ("V50_6" AND ("V15_6" OR "DB22_DisplayData".dbx21_0)) OR ("DB22_DisplayData".dbx21_1 AND NOT "V50_6" AND NOT "V50_7" AND NOT "In_Pos7") OR ("V50_7" AND "DB10_ExtConveyors".Out_ConvPos8);
END_REGION

REGION Network 36: Conveyor pos8 motor
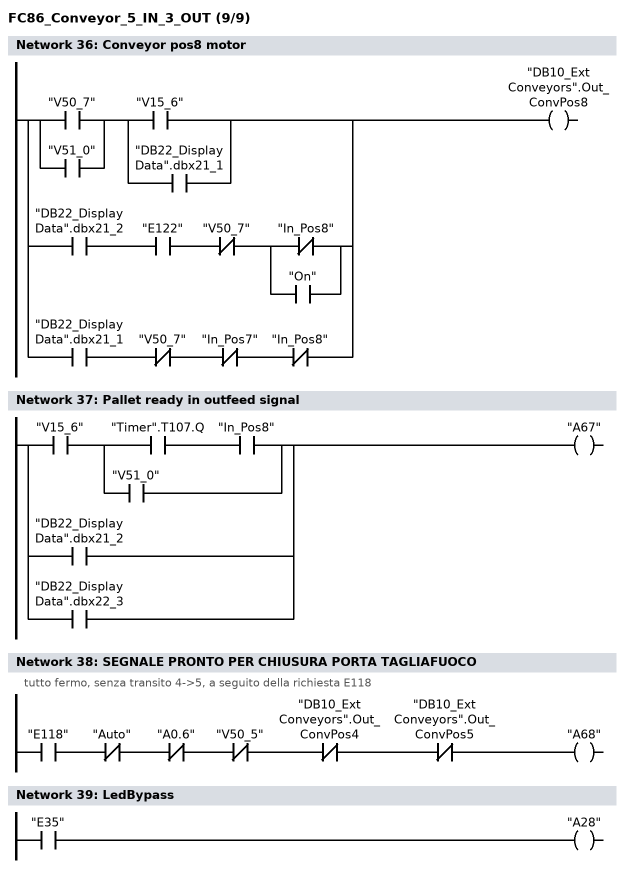
   RUNG wire#powerrail
      Contact( "V50_7" )
      wire#w1
      Contact( "V15_6" )
      wire#w2
      Coil( "DB10_ExtConveyors".Out_ConvPos8 )
   END_RUNG
   RUNG wire#powerrail
      Contact( "V51_0" )
   END_RUNG wire#w1
   RUNG wire#w1
      Contact( "DB22_DisplayData".dbx21_1 )
   END_RUNG wire#w2
   RUNG wire#powerrail
      Contact( "DB22_DisplayData".dbx21_2 )
      Contact( "E122" )
      I_Contact( "V50_7" )
      wire#w3
      I_Contact( "In_Pos8" )
   END_RUNG wire#w2
   RUNG wire#w3
      Contact( "On" )
   END_RUNG wire#w2
   RUNG wire#powerrail
      Contact( "DB22_DisplayData".dbx21_1 )
      I_Contact( "V50_7" )
      I_Contact( "In_Pos7" )
      I_Contact( "In_Pos8" )
   END_RUNG wire#w2
   // the same network as SCL:
   "DB10_ExtConveyors".Out_ConvPos8 := (("V50_7" OR "V51_0") AND ("V15_6" OR "DB22_DisplayData".dbx21_1)) OR ("DB22_DisplayData".dbx21_2 AND "E122" AND NOT "V50_7" AND (NOT "In_Pos8" OR "On")) OR ("DB22_DisplayData".dbx21_1 AND NOT "V50_7" AND NOT "In_Pos7" AND NOT "In_Pos8");
END_REGION

REGION Network 37: Pallet ready in outfeed signal
   RUNG wire#powerrail
      Contact( "V15_6" )
      wire#w1
      Contact( "Timer".T107.Q )
      Contact( "In_Pos8" )
      wire#w2
      Coil( "A67" )
   END_RUNG
   RUNG wire#w1
      Contact( "V51_0" )
   END_RUNG wire#w2
   RUNG wire#powerrail
      Contact( "DB22_DisplayData".dbx21_2 )
   END_RUNG wire#w2
   RUNG wire#powerrail
      Contact( "DB22_DisplayData".dbx22_3 )
   END_RUNG wire#w2
   // the same network as SCL:
   "A67" := ("V15_6" AND (("Timer".T107.Q AND "In_Pos8") OR "V51_0")) OR "DB22_DisplayData".dbx21_2 OR "DB22_DisplayData".dbx22_3;
END_REGION

REGION Network 38: SEGNALE PRONTO PER CHIUSURA PORTA TAGLIAFUOCO
   // tutto fermo, senza transito 4->5, a seguito della richiesta E118
   RUNG wire#powerrail
      Contact( "E118" )
      I_Contact( "Auto" )
      I_Contact( "A0.6" )
      I_Contact( "V50_5" )
      I_Contact( "DB10_ExtConveyors".Out_ConvPos4 )
      I_Contact( "DB10_ExtConveyors".Out_ConvPos5 )
      Coil( "A68" )
   END_RUNG
   // the same network as SCL:
   "A68" := "E118" AND NOT "Auto" AND NOT "A0.6" AND NOT "V50_5" AND NOT "DB10_ExtConveyors".Out_ConvPos4 AND NOT "DB10_ExtConveyors".Out_ConvPos5;
END_REGION

REGION Network 39: LedBypass
   RUNG wire#powerrail
      Contact( "E35" )
      Coil( "A28" )
   END_RUNG
   // the same network as SCL:
   "A28" := "E35";
END_REGION
END_FUNCTION

FUNCTION "FC71_Conveyor_0_IN_0_OUT" : Void   // FC71, LAD
TITLE = Conveyor_0_IN_0_OUT
{ S7_Optimized_Access := 'FALSE' }
VERSION : 0.1
// stored: AutoNumber false, IsIECCheckEnabled false, SetENOAutomatically false, UDAEnableTagReadback false
BEGIN

REGION Network 1: Conveyor manual movement
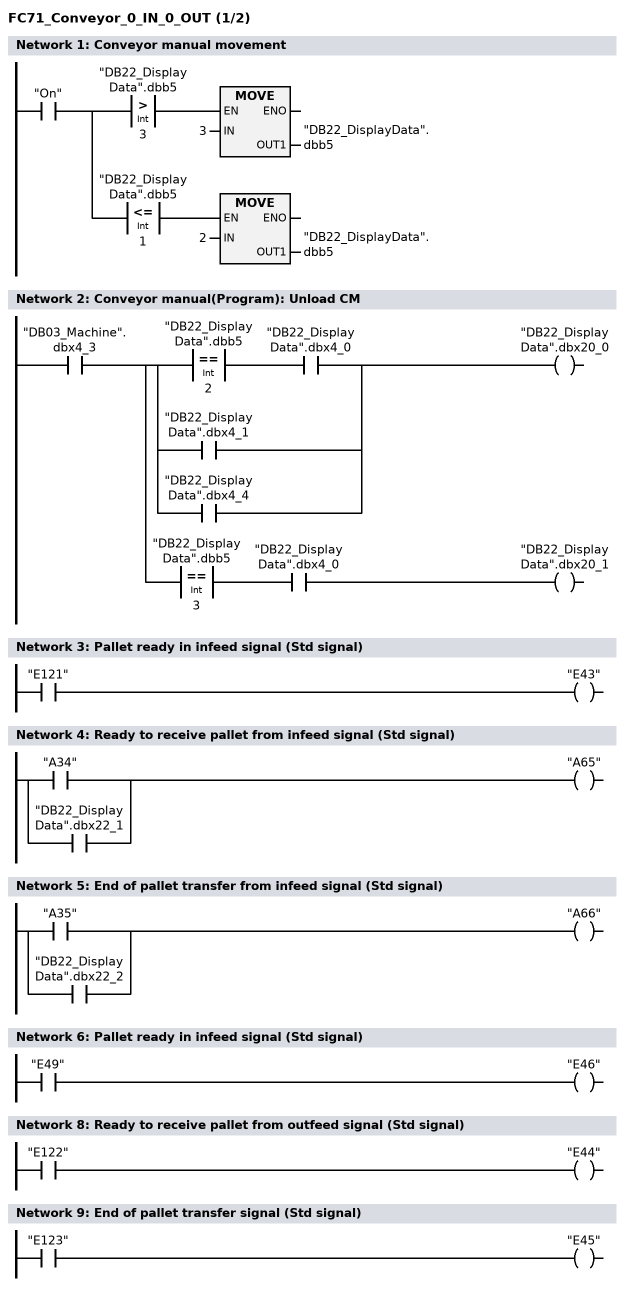
   RUNG wire#powerrail
      Contact( "On" )
      wire#w1
      { S7_Templates := "SrcType := Int" } GT_Contact(in1 := "DB22_DisplayData".dbb5, in2 := 3)
      { S7_GenerateENO := "TRUE" } Move(in := 3, out1 => "DB22_DisplayData".dbb5)
   END_RUNG
   RUNG wire#w1
      { S7_Templates := "SrcType := Int" } LE_Contact(in1 := "DB22_DisplayData".dbb5, in2 := 1)
      { S7_GenerateENO := "TRUE" } Move(in := 2, out1 => "DB22_DisplayData".dbb5)
   END_RUNG
   // the same network as SCL:
   IF "On" AND ("DB22_DisplayData".dbb5 > 3) THEN "DB22_DisplayData".dbb5 := 3; END_IF;
   IF "On" AND ("DB22_DisplayData".dbb5 <= 1) THEN "DB22_DisplayData".dbb5 := 2; END_IF;
END_REGION

REGION Network 2: Conveyor manual(Program): Unload CM
   RUNG wire#powerrail
      Contact( "DB03_Machine".dbx4_3 )
      wire#w1
      { S7_Templates := "SrcType := Int" } EQ_Contact(in1 := "DB22_DisplayData".dbb5, in2 := 2)
      Contact( "DB22_DisplayData".dbx4_0 )
      wire#w2
      Coil( "DB22_DisplayData".dbx20_0 )
   END_RUNG
   RUNG wire#w1
      Contact( "DB22_DisplayData".dbx4_1 )
   END_RUNG wire#w2
   RUNG wire#w1
      Contact( "DB22_DisplayData".dbx4_4 )
   END_RUNG wire#w2
   RUNG wire#w1
      { S7_Templates := "SrcType := Int" } EQ_Contact(in1 := "DB22_DisplayData".dbb5, in2 := 3)
      Contact( "DB22_DisplayData".dbx4_0 )
      Coil( "DB22_DisplayData".dbx20_1 )
   END_RUNG
   // the same network as SCL:
   "DB22_DisplayData".dbx20_0 := "DB03_Machine".dbx4_3 AND ((("DB22_DisplayData".dbb5 = 2) AND "DB22_DisplayData".dbx4_0) OR "DB22_DisplayData".dbx4_1 OR "DB22_DisplayData".dbx4_4);
   "DB22_DisplayData".dbx20_1 := "DB03_Machine".dbx4_3 AND ("DB22_DisplayData".dbb5 = 3) AND "DB22_DisplayData".dbx4_0;
END_REGION

REGION Network 3: Pallet ready in infeed signal (Std signal)
   RUNG wire#powerrail
      Contact( "E121" )
      Coil( "E43" )
   END_RUNG
   // the same network as SCL:
   "E43" := "E121";
END_REGION

REGION Network 4: Ready to receive pallet from infeed signal (Std signal)
   RUNG wire#powerrail
      Contact( "A34" )
      wire#w1
      Coil( "A65" )
   END_RUNG
   RUNG wire#powerrail
      Contact( "DB22_DisplayData".dbx22_1 )
   END_RUNG wire#w1
   // the same network as SCL:
   "A65" := "A34" OR "DB22_DisplayData".dbx22_1;
END_REGION

REGION Network 5: End of pallet transfer from infeed signal (Std signal)
   RUNG wire#powerrail
      Contact( "A35" )
      wire#w1
      Coil( "A66" )
   END_RUNG
   RUNG wire#powerrail
      Contact( "DB22_DisplayData".dbx22_2 )
   END_RUNG wire#w1
   // the same network as SCL:
   "A66" := "A35" OR "DB22_DisplayData".dbx22_2;
END_REGION

REGION Network 6: Pallet ready in infeed signal (Std signal)
   RUNG wire#powerrail
      Contact( "E49" )
      Coil( "E46" )
   END_RUNG
   // the same network as SCL:
   "E46" := "E49";
END_REGION

REGION Network 7: >>>>> OUTFEED CONVEYOR <<<<<<
END_REGION

REGION Network 8: Ready to receive pallet from outfeed signal (Std signal)
   RUNG wire#powerrail
      Contact( "E122" )
      Coil( "E44" )
   END_RUNG
   // the same network as SCL:
   "E44" := "E122";
END_REGION

REGION Network 9: End of pallet transfer signal (Std signal)
   RUNG wire#powerrail
      Contact( "E123" )
      Coil( "E45" )
   END_RUNG
   // the same network as SCL:
   "E45" := "E123";
END_REGION

REGION Network 10: Pallet ready for outfeed signal (Std signal)
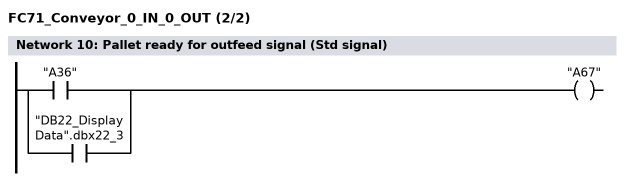
   RUNG wire#powerrail
      Contact( "A36" )
      wire#w1
      Coil( "A67" )
   END_RUNG
   RUNG wire#powerrail
      Contact( "DB22_DisplayData".dbx22_3 )
   END_RUNG wire#w1
   // the same network as SCL:
   "A67" := "A36" OR "DB22_DisplayData".dbx22_3;
END_REGION
END_FUNCTION

FUNCTION "FC72_Conveyor_0_IN_1_OUT" : Void   // FC72, LAD
TITLE = Conveyor_0_IN_1_OUT
{ S7_Optimized_Access := 'FALSE' }
VERSION : 0.1
// stored: AutoNumber false, IsIECCheckEnabled false, SetENOAutomatically false, UDAEnableTagReadback false
   VAR_TEMP   // added for the SCL form of the ladder/FBD networks
      _w1 : Bool;
   END_VAR
BEGIN

REGION Network 1: Conveyor manual movement
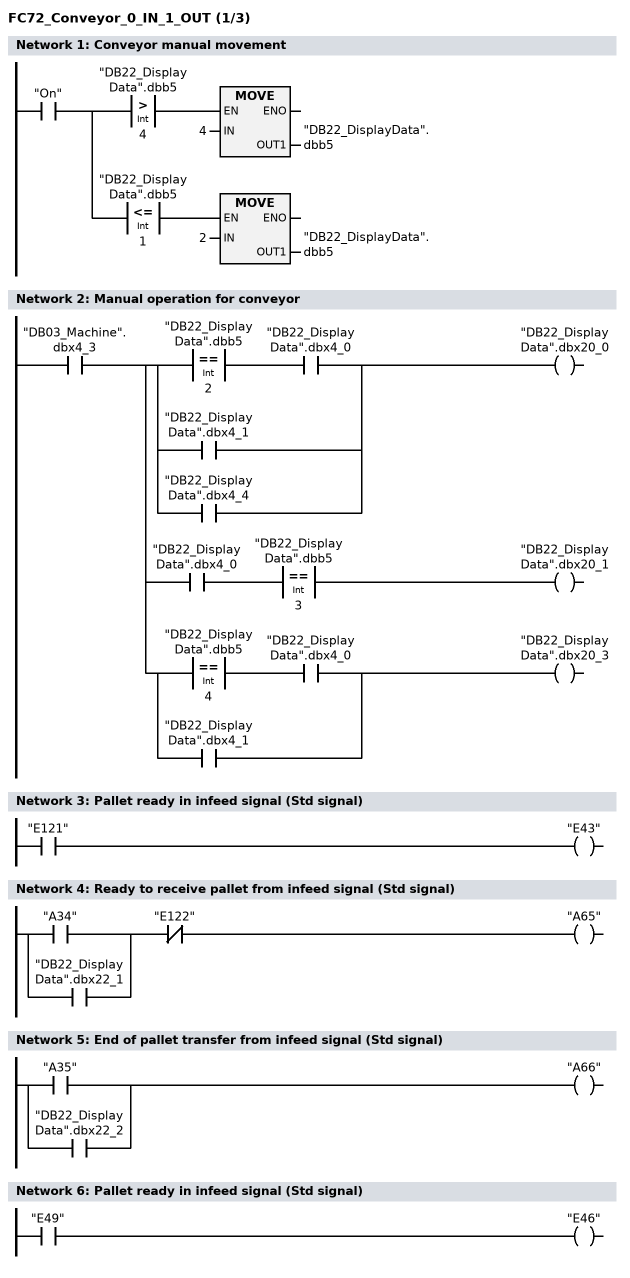
   RUNG wire#powerrail
      Contact( "On" )
      wire#w1
      { S7_Templates := "SrcType := Int" } GT_Contact(in1 := "DB22_DisplayData".dbb5, in2 := 4)
      { S7_GenerateENO := "TRUE" } Move(in := 4, out1 => "DB22_DisplayData".dbb5)
   END_RUNG
   RUNG wire#w1
      { S7_Templates := "SrcType := Int" } LE_Contact(in1 := "DB22_DisplayData".dbb5, in2 := 1)
      { S7_GenerateENO := "TRUE" } Move(in := 2, out1 => "DB22_DisplayData".dbb5)
   END_RUNG
   // the same network as SCL:
   IF "On" AND ("DB22_DisplayData".dbb5 > 4) THEN "DB22_DisplayData".dbb5 := 4; END_IF;
   IF "On" AND ("DB22_DisplayData".dbb5 <= 1) THEN "DB22_DisplayData".dbb5 := 2; END_IF;
END_REGION

REGION Network 2: Manual operation for conveyor
   RUNG wire#powerrail
      Contact( "DB03_Machine".dbx4_3 )
      wire#w1
      { S7_Templates := "SrcType := Int" } EQ_Contact(in1 := "DB22_DisplayData".dbb5, in2 := 2)
      Contact( "DB22_DisplayData".dbx4_0 )
      wire#w2
      Coil( "DB22_DisplayData".dbx20_0 )
   END_RUNG
   RUNG wire#w1
      Contact( "DB22_DisplayData".dbx4_1 )
   END_RUNG wire#w2
   RUNG wire#w1
      Contact( "DB22_DisplayData".dbx4_4 )
   END_RUNG wire#w2
   RUNG wire#w1
      Contact( "DB22_DisplayData".dbx4_0 )
      { S7_Templates := "SrcType := Int" } EQ_Contact(in1 := "DB22_DisplayData".dbb5, in2 := 3)
      Coil( "DB22_DisplayData".dbx20_1 )
   END_RUNG
   RUNG wire#w1
      { S7_Templates := "SrcType := Int" } EQ_Contact(in1 := "DB22_DisplayData".dbb5, in2 := 4)
      Contact( "DB22_DisplayData".dbx4_0 )
      wire#w3
      Coil( "DB22_DisplayData".dbx20_3 )
   END_RUNG
   RUNG wire#w1
      Contact( "DB22_DisplayData".dbx4_1 )
   END_RUNG wire#w3
   // the same network as SCL:
   "DB22_DisplayData".dbx20_0 := "DB03_Machine".dbx4_3 AND ((("DB22_DisplayData".dbb5 = 2) AND "DB22_DisplayData".dbx4_0) OR "DB22_DisplayData".dbx4_1 OR "DB22_DisplayData".dbx4_4);
   "DB22_DisplayData".dbx20_1 := "DB03_Machine".dbx4_3 AND "DB22_DisplayData".dbx4_0 AND ("DB22_DisplayData".dbb5 = 3);
   "DB22_DisplayData".dbx20_3 := "DB03_Machine".dbx4_3 AND ((("DB22_DisplayData".dbb5 = 4) AND "DB22_DisplayData".dbx4_0) OR "DB22_DisplayData".dbx4_1);
END_REGION

REGION Network 3: Pallet ready in infeed signal (Std signal)
   RUNG wire#powerrail
      Contact( "E121" )
      Coil( "E43" )
   END_RUNG
   // the same network as SCL:
   "E43" := "E121";
END_REGION

REGION Network 4: Ready to receive pallet from infeed signal (Std signal)
   RUNG wire#powerrail
      Contact( "A34" )
      wire#w1
      I_Contact( "E122" )
      Coil( "A65" )
   END_RUNG
   RUNG wire#powerrail
      Contact( "DB22_DisplayData".dbx22_1 )
   END_RUNG wire#w1
   // the same network as SCL:
   "A65" := ("A34" OR "DB22_DisplayData".dbx22_1) AND NOT "E122";
END_REGION

REGION Network 5: End of pallet transfer from infeed signal (Std signal)
   RUNG wire#powerrail
      Contact( "A35" )
      wire#w1
      Coil( "A66" )
   END_RUNG
   RUNG wire#powerrail
      Contact( "DB22_DisplayData".dbx22_2 )
   END_RUNG wire#w1
   // the same network as SCL:
   "A66" := "A35" OR "DB22_DisplayData".dbx22_2;
END_REGION

REGION Network 6: Pallet ready in infeed signal (Std signal)
   RUNG wire#powerrail
      Contact( "E49" )
      Coil( "E46" )
   END_RUNG
   // the same network as SCL:
   "E46" := "E49";
END_REGION

REGION Network 7: >>>>> OUTFEED CONVEYOR <<<<<<
END_REGION

REGION Network 8: Time for pallet unload with forklift
